LIN {X 0,Y 601.05,Z 422.346,A -85,B 0,C 180,E1 28225.786,E2 28225.786} C_VEL
LIN {X 0,Y 601.044,Z 422.337,A -85,B 0,C 180,E1 28222.492,E2 28222.492} C_VEL
LIN {X 0,Y 601.04,Z 422.335,A -85,B 0,C 180,E1 28219.923,E2 28219.923} C_VEL
LIN {X 0,Y 601.083,Z 422.357,A -85,B 0,C 180,E1 28216.736,E2 28216.736} C_VEL
LIN {X 0,Y 601.144,Z 422.564,A -85,B 0,C 180,E1 28214.936,E2 28214.936} C_VEL
LIN {X 0,Y 604.045,Z 429.719,A -85,B 0,C 180,E1 28213.94,E2 28213.94} C_VEL
LIN {X 0,Y 612.426,Z 450.093,A -85,B 0,C 180,E1 28211.32,E2 28211.32} C_VEL
LIN {X 0,Y 619.561,Z 469.104,A -85,B 0,C 180,E1 28209.079,E2 28209.079} C_VEL
LIN {X 0,Y 619.97,Z 470.564,A -85,B 0,C 180,E1 28208.923,E2 28208.923} C_VEL
LIN {X 0,Y 618.198,Z 495.68,A -85,B 0,C 180,E1 28206.964,E2 28206.964} C_VEL
LIN {X 0,Y 624.328,Z 523.905,A -85,B 0,C 180,E1 28206.115,E2 28206.115} C_VEL
LIN {X 0,Y 624.389,Z 528.229,A -85,B 0,C 180,E1 28206.051,E2 28206.051} C_VEL
LIN {X 0,Y 622.576,Z 534.727,A -85,B 0,C 180,E1 28206.091,E2 28206.091} C_VEL
LIN {X 0,Y 619.497,Z 543.485,A -85,B 0,C 180,E1 28206.191,E2 28206.191} C_VEL
LIN {X 0,Y 618.976,Z 547.292,A -85,B 0,C 180,E1 28206.176,E2 28206.176} C_VEL
LIN {X 0,Y 614.774,Z 810.927,A -85,B 0,C 180,E1 28202.873,E2 28202.873} C_VEL
LIN {X 0,Y 613.983,Z 851.148,A -85,B 0,C 180,E1 28202.339,E2 28202.339} C_VEL
LIN {X 0,Y 613.023,Z 872.802,A -85,B 0,C 180,E1 28201.895,E2 28201.895} C_VEL
LIN {X 0,Y 611.761,Z 895.07,A -85,B 0,C 180,E1 28201.289,E2 28201.289} C_VEL
LIN {X 0,Y 610.189,Z 916.453,A -85,B 0,C 180,E1 28200.53,E2 28200.53} C_VEL
LIN {X 0,Y 608.411,Z 937.861,A -85,B 0,C 180,E1 28199.6,E2 28199.6} C_VEL
LIN {X 0,Y 606.619,Z 956.702,A -85,B 0,C 180,E1 28198.609,E2 28198.609} C_VEL
LIN {X 0,Y 604.551,Z 976.76,A -85,B 0,C 180,E1 28197.374,E2 28197.374} C_VEL
LIN {X 0,Y 602.523,Z 995.2,A -85,B 0,C 180,E1 28196.036,E2 28196.036} C_VEL
LIN {X 0,Y 600.358,Z 1014.63,A -85,B 0,C 180,E1 28194.396,E2 28194.396} C_VEL
LIN {X 0,Y 598.531,Z 1031.433,A -85,B 0,C 180,E1 28192.756,E2 28192.756} C_VEL
LIN {X 0,Y 596.872,Z 1046.866,A -85,B 0,C 180,E1 28191.008,E2 28191.008} C_VEL
LIN {X 0,Y 595.449,Z 1061.5,A -85,B 0,C 180,E1 28189.114,E2 28189.114} C_VEL
LIN {X 0,Y 594.262,Z 1074.683,A -85,B 0,C 180,E1 28187.117,E2 28187.117} C_VEL
LIN {X 0,Y 593.331,Z 1086.983,A -85,B 0,C 180,E1 28184.942,E2 28184.942} C_VEL
LIN {X 0,Y 592.724,Z 1096.907,A -85,B 0,C 180,E1 28182.866,E2 28182.866} C_VEL
LIN {X 0,Y 592.299,Z 1105.822,A -85,B 0,C 180,E1 28180.603,E2 28180.603} C_VEL
LIN {X 0,Y 592.042,Z 1113.446,A -85,B 0,C 180,E1 28178.156,E2 28178.156} C_VEL
LIN {X 0,Y 591.953,Z 1118.281,A -85,B 0,C 180,E1 28176.109,E2 28176.109} C_VEL
LIN {X 0,Y 591.903,Z 1122.06,A -85,B 0,C 180,E1 28173.778,E2 28173.778} C_VEL
LIN {X 0,Y 591.898,Z 1123.925,A -85,B 0,C 180,E1 28171.742,E2 28171.742} C_VEL
LIN {X 0,Y 591.894,Z 1124.401,A -85,B 0,C 180,E1 28169.516,E2 28169.516} C_VEL
LIN {X 0,Y 591.895,Z 1123.448,A -85,B 0,C 180,E1 28167.483,E2 28167.483} C_VEL
LIN {X 0,Y 591.909,Z 1120.693,A -85,B 0,C 180,E1 28165.155,E2 28165.155} C_VEL
LIN {X 0,Y 591.961,Z 1116.818,A -85,B 0,C 180,E1 28163.112,E2 28163.112} C_VEL
LIN {X 0,Y 592.104,Z 1110.894,A -85,B 0,C 180,E1 28160.866,E2 28160.866} C_VEL
LIN {X 0,Y 592.394,Z 1103.29,A -85,B 0,C 180,E1 28158.61,E2 28158.61} C_VEL
LIN {X 0,Y 592.842,Z 1094.611,A -85,B 0,C 180,E1 28156.541,E2 28156.541} C_VEL
LIN {X 0,Y 593.533,Z 1084.376,A -85,B 0,C 180,E1 28154.463,E2 28154.463} C_VEL
LIN {X 0,Y 594.419,Z 1072.701,A -85,B 0,C 180,E1 28152.476,E2 28152.476} C_VEL
LIN {X 0,Y 595.654,Z 1059.219,A -85,B 0,C 180,E1 28150.485,E2 28150.485} C_VEL
LIN {X 0,Y 597.056,Z 1045.112,A -85,B 0,C 180,E1 28148.69,E2 28148.69} C_VEL
LIN {X 0,Y 598.825,Z 1028.383,A -85,B 0,C 180,E1 28146.844,E2 28146.844} C_VEL
LIN {X 0,Y 600.769,Z 1011.25,A -85,B 0,C 180,E1 28145.202,E2 28145.202} C_VEL
LIN {X 0,Y 602.748,Z 993.069,A -85,B 0,C 180,E1 28143.709,E2 28143.709} C_VEL
LIN {X 0,Y 604.798,Z 974.681,A -85,B 0,C 180,E1 28142.394,E2 28142.394} C_VEL
LIN {X 0,Y 606.783,Z 955.027,A -85,B 0,C 180,E1 28141.206,E2 28141.206} C_VEL
LIN {X 0,Y 608.708,Z 934.494,A -85,B 0,C 180,E1 28140.149,E2 28140.149} C_VEL
LIN {X 0,Y 610.427,Z 913.492,A -85,B 0,C 180,E1 28139.265,E2 28139.265} C_VEL
LIN {X 0,Y 612.059,Z 890.14,A -85,B 0,C 180,E1 28138.475,E2 28138.475} C_VEL
LIN {X 0,Y 613.177,Z 869.724,A -85,B 0,C 180,E1 28137.941,E2 28137.941} C_VEL
LIN {X 0,Y 614.133,Z 844.992,A -85,B 0,C 180,E1 28137.477,E2 28137.477} C_VEL
LIN {X 0,Y 617.7,Z 621.355,A -85,B 0,C 180,E1 28134.667,E2 28134.667} C_VEL
LIN {X 0,Y 619.107,Z 530.98,A -85,B 0,C 180,E1 28133.514,E2 28133.514} C_VEL
LIN {X 0,Y 611.434,Z 494.69,A -85,B 0,C 180,E1 28132.397,E2 28132.397} C_VEL
LIN {X 0,Y 613.03,Z 473.555,A -85,B 0,C 180,E1 28130.709,E2 28130.709} C_VEL
LIN {X 0,Y 605.976,Z 454.567,A -85,B 0,C 180,E1 28128.446,E2 28128.446} C_VEL
LIN {X 0,Y 597.834,Z 434.608,A -85,B 0,C 180,E1 28125.85,E2 28125.85} C_VEL
LIN {X 0,Y 593.852,Z 425.716,A -85,B 0,C 180,E1 28124.597,E2 28124.597} C_VEL
LIN {X 0,Y 593.146,Z 423.487,A -85,B 0,C 180,E1 28124.238,E2 28124.238} C_VEL
LIN {X 0,Y 593.126,Z 423.302,A -85,B 0,C 180,E1 28121.364,E2 28121.364} C_VEL
LIN {X 0,Y 593.115,Z 423.346,A -85,B 0,C 180,E1 28118.067,E2 28118.067} C_VEL
LIN {X 0,Y 593.129,Z 423.304,A -85,B 0,C 180,E1 28115.154,E2 28115.154} C_VEL
LIN {X 0,Y 593.105,Z 423.34,A -85,B 0,C 180,E1 28111.962,E2 28111.962} C_VEL
LIN {X 0,Y 593.118,Z 423.349,A -85,B 0,C 180,E1 28109.157,E2 28109.157} C_VEL
LIN {X 0,Y 593.103,Z 423.347,A -85,B 0,C 180,E1 28105.89,E2 28105.89} C_VEL
LIN {X 0,Y 593.124,Z 423.346,A -85,B 0,C 180,E1 28103.008,E2 28103.008} C_VEL
LIN {X 0,Y 593.113,Z 423.346,A -85,B 0,C 180,E1 28099.807,E2 28099.807} C_VEL
LIN {X 0,Y 593.124,Z 423.335,A -85,B 0,C 180,E1 28096.956,E2 28096.956} C_VEL
LIN {X 0,Y 593.122,Z 423.341,A -85,B 0,C 180,E1 28093.751,E2 28093.751} C_VEL
LIN {X 0,Y 593.131,Z 423.343,A -85,B 0,C 180,E1 28090.883,E2 28090.883} C_VEL
LIN {X 0,Y 593.124,Z 423.336,A -85,B 0,C 180,E1 28087.556,E2 28087.556} C_VEL
LIN {X 0,Y 593.143,Z 423.34,A -85,B 0,C 180,E1 28084.738,E2 28084.738} C_VEL
LIN {X 0,Y 593.131,Z 423.344,A -85,B 0,C 180,E1 28081.449,E2 28081.449} C_VEL
LIN {X 0,Y 593.157,Z 423.328,A -85,B 0,C 180,E1 28078.551,E2 28078.551} C_VEL
LIN {X 0,Y 593.137,Z 423.334,A -85,B 0,C 180,E1 28075.359,E2 28075.359} C_VEL
LIN {X 0,Y 593.176,Z 423.345,A -85,B 0,C 180,E1 28072.347,E2 28072.347} C_VEL
LIN {X 0,Y 593.14,Z 423.337,A -85,B 0,C 180,E1 28069.117,E2 28069.117} C_VEL
LIN {X 0,Y 593.198,Z 423.324,A -85,B 0,C 180,E1 28066.052,E2 28066.052} C_VEL
LIN {X 0,Y 593.145,Z 423.341,A -85,B 0,C 180,E1 28062.906,E2 28062.906} C_VEL
LIN {X 0,Y 593.201,Z 423.339,A -85,B 0,C 180,E1 28059.785,E2 28059.785} C_VEL
LIN {X 0,Y 593.153,Z 423.338,A -85,B 0,C 180,E1 28056.663,E2 28056.663} C_VEL
LIN {X 0,Y 593.198,Z 423.333,A -85,B 0,C 180,E1 28053.469,E2 28053.469} C_VEL
LIN {X 0,Y 593.168,Z 423.332,A -85,B 0,C 180,E1 28050.291,E2 28050.291} C_VEL
LIN {X 0,Y 593.171,Z 423.302,A -85,B 0,C 180,E1 28047.011,E2 28047.011} C_VEL
LIN {X 0,Y 593.194,Z 423.336,A -85,B 0,C 180,E1 28043.844,E2 28043.844} C_VEL
LIN {X 0,Y 593.16,Z 423.296,A -85,B 0,C 180,E1 28040.667,E2 28040.667} C_VEL
LIN {X 0,Y 593.194,Z 423.319,A -85,B 0,C 180,E1 28037.587,E2 28037.587} C_VEL
LIN {X 0,Y 593.202,Z 423.558,A -85,B 0,C 180,E1 28036.492,E2 28036.492} C_VEL
LIN {X 0,Y 596.23,Z 430.677,A -85,B 0,C 180,E1 28035.493,E2 28035.493} C_VEL
LIN {X 0,Y 604.145,Z 449.031,A -85,B 0,C 180,E1 28033.121,E2 28033.121} C_VEL
LIN {X 0,Y 607.608,Z 457.418,A -85,B 0,C 180,E1 28032.136,E2 28032.136} C_VEL
LIN {X 0,Y 620.44,Z 478.904,A -85,B 0,C 180,E1 28030.804,E2 28030.804} C_VEL
LIN {X 0,Y 622.327,Z 489.051,A -85,B 0,C 180,E1 28030.513,E2 28030.513} C_VEL
LIN {X 0,Y 617.253,Z 739.769,A -85,B 0,C 180,E1 28027.182,E2 28027.182} C_VEL
LIN {X 0,Y 615.172,Z 843.964,A -85,B 0,C 180,E1 28025.791,E2 28025.791} C_VEL
LIN {X 0,Y 614.103,Z 869.036,A -85,B 0,C 180,E1 28025.297,E2 28025.297} C_VEL
LIN {X 0,Y 612.948,Z 889.774,A -85,B 0,C 180,E1 28024.756,E2 28024.756} C_VEL
LIN {X 0,Y 611.336,Z 914.776,A -85,B 0,C 180,E1 28023.93,E2 28023.93} C_VEL
LIN {X 0,Y 609.706,Z 936.084,A -85,B 0,C 180,E1 28023.068,E2 28023.068} C_VEL
LIN {X 0,Y 607.878,Z 958.694,A -85,B 0,C 180,E1 28021.982,E2 28021.982} C_VEL
LIN {X 0,Y 606.11,Z 978.363,A -85,B 0,C 180,E1 28020.868,E2 28020.868} C_VEL
LIN {X 0,Y 604.212,Z 998.769,A -85,B 0,C 180,E1 28019.548,E2 28019.548} C_VEL
LIN {X 0,Y 602.242,Z 1018.444,A -85,B 0,C 180,E1 28018.065,E2 28018.065} C_VEL
LIN {X 0,Y 600.563,Z 1035.551,A -85,B 0,C 180,E1 28016.607,E2 28016.607} C_VEL
LIN {X 0,Y 598.715,Z 1054.222,A -85,B 0,C 180,E1 28014.783,E2 28014.783} C_VEL
LIN {X 0,Y 597.317,Z 1068.791,A -85,B 0,C 180,E1 28013.165,E2 28013.165} C_VEL
LIN {X 0,Y 595.868,Z 1084.777,A -85,B 0,C 180,E1 28011.148,E2 28011.148} C_VEL
LIN {X 0,Y 594.797,Z 1097.221,A -85,B 0,C 180,E1 28009.34,E2 28009.34} C_VEL
LIN {X 0,Y 593.82,Z 1109.687,A -85,B 0,C 180,E1 28007.239,E2 28007.239} C_VEL
LIN {X 0,Y 593.064,Z 1120.636,A -85,B 0,C 180,E1 28005.049,E2 28005.049} C_VEL
LIN {X 0,Y 592.573,Z 1129.582,A -85,B 0,C 180,E1 28002.969,E2 28002.969} C_VEL
LIN {X 0,Y 592.216,Z 1137.906,A -85,B 0,C 180,E1 28000.605,E2 28000.605} C_VEL
LIN {X 0,Y 592.035,Z 1143.491,A -85,B 0,C 180,E1 27998.645,E2 27998.645} C_VEL
LIN {X 0,Y 591.95,Z 1148.695,A -85,B 0,C 180,E1 27996.304,E2 27996.304} C_VEL
LIN {X 0,Y 591.92,Z 1152.008,A -85,B 0,C 180,E1 27994.068,E2 27994.068} C_VEL
LIN {X 0,Y 591.908,Z 1153.903,A -85,B 0,C 180,E1 27991.936,E2 27991.936} C_VEL
LIN {X 0,Y 591.885,Z 1154.394,A -85,B 0,C 180,E1 27989.516,E2 27989.516} C_VEL
LIN {X 0,Y 591.897,Z 1153.494,A -85,B 0,C 180,E1 27987.483,E2 27987.483} C_VEL
LIN {X 0,Y 591.911,Z 1151.085,A -85,B 0,C 180,E1 27985.155,E2 27985.155} C_VEL
LIN {X 0,Y 591.973,Z 1147.102,A -85,B 0,C 180,E1 27982.917,E2 27982.917} C_VEL
LIN {X 0,Y 592.066,Z 1142.219,A -85,B 0,C 180,E1 27980.866,E2 27980.866} C_VEL
LIN {X 0,Y 592.321,Z 1134.659,A -85,B 0,C 180,E1 27978.411,E2 27978.411} C_VEL
LIN {X 0,Y 592.678,Z 1127.151,A -85,B 0,C 180,E1 27976.438,E2 27976.438} C_VEL
LIN {X 0,Y 593.285,Z 1117.27,A -85,B 0,C 180,E1 27974.225,E2 27974.225} C_VEL
LIN {X 0,Y 594.113,Z 1105.682,A -85,B 0,C 180,E1 27972.062,E2 27972.062} C_VEL
LIN {X 0,Y 595.031,Z 1094.406,A -85,B 0,C 180,E1 27970.225,E2 27970.225} C_VEL
LIN {X 0,Y 596.331,Z 1079.433,A -85,B 0,C 180,E1 27968.146,E2 27968.146} C_VEL
LIN {X 0,Y 597.651,Z 1065.334,A -85,B 0,C 180,E1 27966.431,E2 27966.431} C_VEL
LIN {X 0,Y 599.431,Z 1047.001,A -85,B 0,C 180,E1 27964.479,E2 27964.479} C_VEL
LIN {X 0,Y 601.065,Z 1030.416,A -85,B 0,C 180,E1 27962.936,E2 27962.936} C_VEL
LIN {X 0,Y 603.114,Z 1009.862,A -85,B 0,C 180,E1 27961.263,E2 27961.263} C_VEL
LIN {X 0,Y 604.896,Z 991.183,A -85,B 0,C 180,E1 27959.943,E2 27959.943} C_VEL
LIN {X 0,Y 606.901,Z 969.837,A -85,B 0,C 180,E1 27958.626,E2 27958.626} C_VEL
LIN {X 0,Y 608.666,Z 949.321,A -85,B 0,C 180,E1 27957.549,E2 27957.549} C_VEL
LIN {X 0,Y 610.346,Z 928.452,A -85,B 0,C 180,E1 27956.602,E2 27956.602} C_VEL
LIN {X 0,Y 611.969,Z 905.031,A -85,B 0,C 180,E1 27955.725,E2 27955.725} C_VEL
LIN {X 0,Y 613.339,Z 882.784,A -85,B 0,C 180,E1 27955.043,E2 27955.043} C_VEL
LIN {X 0,Y 614.638,Z 857.534,A -85,B 0,C 180,E1 27954.456,E2 27954.456} C_VEL
LIN {X 0,Y 615.43,Z 835.19,A -85,B 0,C 180,E1 27954.079,E2 27954.079} C_VEL
LIN {X 0,Y 620.145,Z 592.09,A -85,B 0,C 180,E1 27950.858,E2 27950.858} C_VEL
LIN {X 0,Y 622.173,Z 487.31,A -85,B 0,C 180,E1 27949.452,E2 27949.452} C_VEL
LIN {X 0,Y 620.052,Z 478.166,A -85,B 0,C 180,E1 27949.158,E2 27949.158} C_VEL
LIN {X 0,Y 607.39,Z 457,A -85,B 0,C 180,E1 27947.835,E2 27947.835} C_VEL
LIN {X 0,Y 599.631,Z 438.401,A -85,B 0,C 180,E1 27945.537,E2 27945.537} C_VEL
LIN {X 0,Y 594.136,Z 426.221,A -85,B 0,C 180,E1 27943.898,E2 27943.898} C_VEL
LIN {X 0,Y 593.189,Z 423.473,A -85,B 0,C 180,E1 27943.481,E2 27943.481} C_VEL
LIN {X 0,Y 593.196,Z 423.3,A -85,B 0,C 180,E1 27940.21,E2 27940.21} C_VEL
LIN {X 0,Y 593.185,Z 423.342,A -85,B 0,C 180,E1 27936.966,E2 27936.966} C_VEL
LIN {X 0,Y 593.163,Z 423.294,A -85,B 0,C 180,E1 27933.683,E2 27933.683} C_VEL
LIN {X 0,Y 593.2,Z 423.341,A -85,B 0,C 180,E1 27930.488,E2 27930.488} C_VEL
LIN {X 0,Y 593.157,Z 423.342,A -85,B 0,C 180,E1 27927.291,E2 27927.291} C_VEL
LIN {X 0,Y 593.2,Z 423.34,A -85,B 0,C 180,E1 27924.074,E2 27924.074} C_VEL
LIN {X 0,Y 593.156,Z 423.339,A -85,B 0,C 180,E1 27920.939,E2 27920.939} C_VEL
LIN {X 0,Y 593.172,Z 423.331,A -85,B 0,C 180,E1 27917.663,E2 27917.663} C_VEL
LIN {X 0,Y 593.162,Z 423.331,A -85,B 0,C 180,E1 27914.626,E2 27914.626} C_VEL
LIN {X 0,Y 593.153,Z 423.339,A -85,B 0,C 180,E1 27911.375,E2 27911.375} C_VEL
LIN {X 0,Y 593.177,Z 423.336,A -85,B 0,C 180,E1 27908.317,E2 27908.317} C_VEL
LIN {X 0,Y 593.138,Z 423.332,A -85,B 0,C 180,E1 27905.126,E2 27905.126} C_VEL
LIN {X 0,Y 593.189,Z 423.336,A -85,B 0,C 180,E1 27902.029,E2 27902.029} C_VEL
LIN {X 0,Y 593.132,Z 423.345,A -85,B 0,C 180,E1 27898.937,E2 27898.937} C_VEL
LIN {X 0,Y 593.19,Z 423.323,A -85,B 0,C 180,E1 27895.843,E2 27895.843} C_VEL
LIN {X 0,Y 593.121,Z 423.337,A -85,B 0,C 180,E1 27892.736,E2 27892.736} C_VEL
LIN {X 0,Y 593.192,Z 423.343,A -85,B 0,C 180,E1 27889.609,E2 27889.609} C_VEL
LIN {X 0,Y 593.115,Z 423.34,A -85,B 0,C 180,E1 27886.547,E2 27886.547} C_VEL
LIN {X 0,Y 593.188,Z 423.328,A -85,B 0,C 180,E1 27883.55,E2 27883.55} C_VEL
LIN {X 0,Y 593.11,Z 423.345,A -85,B 0,C 180,E1 27880.457,E2 27880.457} C_VEL
LIN {X 0,Y 593.188,Z 423.342,A -85,B 0,C 180,E1 27877.398,E2 27877.398} C_VEL
LIN {X 0,Y 593.103,Z 423.345,A -85,B 0,C 180,E1 27874.325,E2 27874.325} C_VEL
LIN {X 0,Y 593.163,Z 423.335,A -85,B 0,C 180,E1 27871.177,E2 27871.177} C_VEL
LIN {X 0,Y 593.093,Z 423.339,A -85,B 0,C 180,E1 27868.264,E2 27868.264} C_VEL
LIN {X 0,Y 593.159,Z 423.309,A -85,B 0,C 180,E1 27865.148,E2 27865.148} C_VEL
LIN {X 0,Y 593.097,Z 423.339,A -85,B 0,C 180,E1 27862.092,E2 27862.092} C_VEL
LIN {X 0,Y 593.171,Z 423.297,A -85,B 0,C 180,E1 27859.025,E2 27859.025} C_VEL
LIN {X 0,Y 593.105,Z 423.337,A -85,B 0,C 180,E1 27856.006,E2 27856.006} C_VEL
LIN {X 0,Y 593.191,Z 423.746,A -85,B 0,C 180,E1 27855.582,E2 27855.582} C_VEL
LIN {X 0,Y 601.081,Z 442.504,A -85,B 0,C 180,E1 27853.003,E2 27853.003} C_VEL
LIN {X 0,Y 607.647,Z 459.038,A -85,B 0,C 180,E1 27850.913,E2 27850.913} C_VEL
LIN {X 0,Y 613.042,Z 474.205,A -85,B 0,C 180,E1 27849.14,E2 27849.14} C_VEL
LIN {X 0,Y 611.468,Z 495.318,A -85,B 0,C 180,E1 27847.48,E2 27847.48} C_VEL
LIN {X 0,Y 619.238,Z 532.257,A -85,B 0,C 180,E1 27846.367,E2 27846.367} C_VEL
LIN {X 0,Y 618.976,Z 547.292,A -85,B 0,C 180,E1 27846.176,E2 27846.176} C_VEL
LIN {X 0,Y 618.033,Z 554.991,A -85,B 0,C 180,E1 27846.136,E2 27846.136} C_VEL
LIN {X 0,Y 612.713,Z 575.535,A -85,B 0,C 180,E1 27846.236,E2 27846.236} C_VEL
LIN {X 0,Y 612.009,Z 582.141,A -85,B 0,C 180,E1 27846.195,E2 27846.195} C_VEL
LIN {X 0,Y 607.943,Z 828.787,A -85,B 0,C 180,E1 27843.084,E2 27843.084} C_VEL
LIN {X 0,Y 607.185,Z 856.005,A -85,B 0,C 180,E1 27842.679,E2 27842.679} C_VEL
LIN {X 0,Y 606.22,Z 876.458,A -85,B 0,C 180,E1 27842.237,E2 27842.237} C_VEL
LIN {X 0,Y 604.704,Z 899.838,A -85,B 0,C 180,E1 27841.557,E2 27841.557} C_VEL
LIN {X 0,Y 603.091,Z 921.266,A -85,B 0,C 180,E1 27840.762,E2 27840.762} C_VEL
LIN {X 0,Y 601.196,Z 941.808,A -85,B 0,C 180,E1 27839.821,E2 27839.821} C_VEL
LIN {X 0,Y 599.287,Z 961.134,A -85,B 0,C 180,E1 27838.774,E2 27838.774} C_VEL
LIN {X 0,Y 597.129,Z 980.515,A -85,B 0,C 180,E1 27837.527,E2 27837.527} C_VEL
LIN {X 0,Y 595.111,Z 998.251,A -85,B 0,C 180,E1 27836.205,E2 27836.205} C_VEL
LIN {X 0,Y 592.941,Z 1016.199,A -85,B 0,C 180,E1 27834.642,E2 27834.642} C_VEL
LIN {X 0,Y 591.03,Z 1032.627,A -85,B 0,C 180,E1 27833.004,E2 27833.004} C_VEL
LIN {X 0,Y 589.218,Z 1048.24,A -85,B 0,C 180,E1 27831.19,E2 27831.19} C_VEL
LIN {X 0,Y 587.627,Z 1063.346,A -85,B 0,C 180,E1 27829.172,E2 27829.172} C_VEL
LIN {X 0,Y 586.448,Z 1075.686,A -85,B 0,C 180,E1 27827.258,E2 27827.258} C_VEL
LIN {X 0,Y 585.481,Z 1087.333,A -85,B 0,C 180,E1 27825.147,E2 27825.147} C_VEL
LIN {X 0,Y 584.821,Z 1097.227,A -85,B 0,C 180,E1 27823.043,E2 27823.043} C_VEL
LIN {X 0,Y 584.358,Z 1105.737,A -85,B 0,C 180,E1 27820.835,E2 27820.835} C_VEL
LIN {X 0,Y 584.091,Z 1112.836,A -85,B 0,C 180,E1 27818.565,E2 27818.565} C_VEL
LIN {X 0,Y 583.959,Z 1117.726,A -85,B 0,C 180,E1 27816.489,E2 27816.489} C_VEL
LIN {X 0,Y 583.915,Z 1121.617,A -85,B 0,C 180,E1 27814.223,E2 27814.223} C_VEL
LIN {X 0,Y 583.907,Z 1123.814,A -85,B 0,C 180,E1 27811.963,E2 27811.963} C_VEL
LIN {X 0,Y 583.896,Z 1124.423,A -85,B 0,C 180,E1 27809.608,E2 27809.608} C_VEL
LIN {X 0,Y 583.896,Z 1123.546,A -85,B 0,C 180,E1 27807.546,E2 27807.546} C_VEL
LIN {X 0,Y 583.907,Z 1121.046,A -85,B 0,C 180,E1 27805.285,E2 27805.285} C_VEL
LIN {X 0,Y 583.961,Z 1117.301,A -85,B 0,C 180,E1 27803.215,E2 27803.215} C_VEL
LIN {X 0,Y 584.112,Z 1111.675,A -85,B 0,C 180,E1 27800.939,E2 27800.939} C_VEL
LIN {X 0,Y 584.384,Z 1104.957,A -85,B 0,C 180,E1 27798.852,E2 27798.852} C_VEL
LIN {X 0,Y 584.895,Z 1095.828,A -85,B 0,C 180,E1 27796.556,E2 27796.556} C_VEL
LIN {X 0,Y 585.614,Z 1085.762,A -85,B 0,C 180,E1 27794.451,E2 27794.451} C_VEL
LIN {X 0,Y 586.614,Z 1073.704,A -85,B 0,C 180,E1 27792.331,E2 27792.331} C_VEL
LIN {X 0,Y 587.932,Z 1060.467,A -85,B 0,C 180,E1 27790.322,E2 27790.322} C_VEL
LIN {X 0,Y 589.413,Z 1046.487,A -85,B 0,C 180,E1 27788.504,E2 27788.504} C_VEL
LIN {X 0,Y 591.259,Z 1030.422,A -85,B 0,C 180,E1 27786.676,E2 27786.676} C_VEL
LIN {X 0,Y 593.201,Z 1014.112,A -85,B 0,C 180,E1 27785.074,E2 27785.074} C_VEL
LIN {X 0,Y 595.475,Z 994.847,A -85,B 0,C 180,E1 27783.439,E2 27783.439} C_VEL
LIN {X 0,Y 597.502,Z 977.421,A -85,B 0,C 180,E1 27782.167,E2 27782.167} C_VEL
LIN {X 0,Y 599.666,Z 957.308,A -85,B 0,C 180,E1 27780.918,E2 27780.918} C_VEL
LIN {X 0,Y 601.526,Z 938.496,A -85,B 0,C 180,E1 27779.922,E2 27779.922} C_VEL
LIN {X 0,Y 603.405,Z 917.009,A -85,B 0,C 180,E1 27778.979,E2 27778.979} C_VEL
LIN {X 0,Y 604.985,Z 896.363,A -85,B 0,C 180,E1 27778.237,E2 27778.237} C_VEL
LIN {X 0,Y 606.369,Z 873.599,A -85,B 0,C 180,E1 27777.604,E2 27777.604} C_VEL
LIN {X 0,Y 607.34,Z 852.734,A -85,B 0,C 180,E1 27777.169,E2 27777.169} C_VEL
LIN {X 0,Y 608.099,Z 819.646,A -85,B 0,C 180,E1 27776.711,E2 27776.711} C_VEL
LIN {X 0,Y 612.468,Z 559.419,A -85,B 0,C 180,E1 27773.426,E2 27773.426} C_VEL
LIN {X 0,Y 612.791,Z 532.472,A -85,B 0,C 180,E1 27773.066,E2 27773.066} C_VEL
LIN {X 0,Y 604.761,Z 494.235,A -85,B 0,C 180,E1 27771.864,E2 27771.864} C_VEL
LIN {X 0,Y 606.055,Z 476.769,A -85,B 0,C 180,E1 27770.443,E2 27770.443} C_VEL
LIN {X 0,Y 599.286,Z 458.457,A -85,B 0,C 180,E1 27768.229,E2 27768.229} C_VEL
LIN {X 0,Y 591.613,Z 439.49,A -85,B 0,C 180,E1 27765.732,E2 27765.732} C_VEL
LIN {X 0,Y 586.509,Z 427.857,A -85,B 0,C 180,E1 27764.073,E2 27764.073} C_VEL
LIN {X 0,Y 585.209,Z 424.511,A -85,B 0,C 180,E1 27763.554,E2 27763.554} C_VEL
LIN {X 0,Y 585.206,Z 424.291,A -85,B 0,C 180,E1 27760.487,E2 27760.487} C_VEL
LIN {X 0,Y 585.166,Z 424.319,A -85,B 0,C 180,E1 27757.707,E2 27757.707} C_VEL
LIN {X 0,Y 585.222,Z 424.301,A -85,B 0,C 180,E1 27754.558,E2 27754.558} C_VEL
LIN {X 0,Y 585.162,Z 424.327,A -85,B 0,C 180,E1 27751.525,E2 27751.525} C_VEL
LIN {X 0,Y 585.203,Z 424.323,A -85,B 0,C 180,E1 27748.359,E2 27748.359} C_VEL
LIN {X 0,Y 585.159,Z 424.335,A -85,B 0,C 180,E1 27745.398,E2 27745.398} C_VEL
LIN {X 0,Y 585.197,Z 424.331,A -85,B 0,C 180,E1 27742.167,E2 27742.167} C_VEL
LIN {X 0,Y 585.17,Z 424.335,A -85,B 0,C 180,E1 27739.256,E2 27739.256} C_VEL
LIN {X 0,Y 585.196,Z 424.328,A -85,B 0,C 180,E1 27735.968,E2 27735.968} C_VEL
LIN {X 0,Y 585.178,Z 424.327,A -85,B 0,C 180,E1 27733.104,E2 27733.104} C_VEL
LIN {X 0,Y 585.201,Z 424.33,A -85,B 0,C 180,E1 27729.838,E2 27729.838} C_VEL
LIN {X 0,Y 585.19,Z 424.326,A -85,B 0,C 180,E1 27726.91,E2 27726.91} C_VEL
LIN {X 0,Y 585.191,Z 424.317,A -85,B 0,C 180,E1 27723.527,E2 27723.527} C_VEL
LIN {X 0,Y 585.217,Z 424.331,A -85,B 0,C 180,E1 27720.587,E2 27720.587} C_VEL
LIN {X 0,Y 585.196,Z 424.332,A -85,B 0,C 180,E1 27717.356,E2 27717.356} C_VEL
LIN {X 0,Y 585.25,Z 424.314,A -85,B 0,C 180,E1 27714.215,E2 27714.215} C_VEL
LIN {X 0,Y 585.199,Z 424.328,A -85,B 0,C 180,E1 27711.154,E2 27711.154} C_VEL
LIN {X 0,Y 585.262,Z 424.329,A -85,B 0,C 180,E1 27707.97,E2 27707.97} C_VEL
LIN {X 0,Y 585.203,Z 424.324,A -85,B 0,C 180,E1 27704.846,E2 27704.846} C_VEL
LIN {X 0,Y 585.256,Z 424.312,A -85,B 0,C 180,E1 27701.678,E2 27701.678} C_VEL
LIN {X 0,Y 585.217,Z 424.325,A -85,B 0,C 180,E1 27698.553,E2 27698.553} C_VEL
LIN {X 0,Y 585.238,Z 424.324,A -85,B 0,C 180,E1 27695.254,E2 27695.254} C_VEL
LIN {X 0,Y 585.255,Z 424.328,A -85,B 0,C 180,E1 27692.041,E2 27692.041} C_VEL
LIN {X 0,Y 585.225,Z 424.332,A -85,B 0,C 180,E1 27688.822,E2 27688.822} C_VEL
LIN {X 0,Y 585.253,Z 424.279,A -85,B 0,C 180,E1 27685.609,E2 27685.609} C_VEL
LIN {X 0,Y 585.225,Z 424.316,A -85,B 0,C 180,E1 27682.414,E2 27682.414} C_VEL
LIN {X 0,Y 585.258,Z 424.302,A -85,B 0,C 180,E1 27679.187,E2 27679.187} C_VEL
LIN {X 0,Y 585.292,Z 424.566,A -85,B 0,C 180,E1 27677.198,E2 27677.198} C_VEL
LIN {X 0,Y 588.532,Z 432.056,A -85,B 0,C 180,E1 27676.118,E2 27676.118} C_VEL
LIN {X 0,Y 596.656,Z 450.909,A -85,B 0,C 180,E1 27673.618,E2 27673.618} C_VEL
LIN {X 0,Y 599.594,Z 457.875,A -85,B 0,C 180,E1 27672.78,E2 27672.78} C_VEL
LIN {X 0,Y 614.47,Z 482.491,A -85,B 0,C 180,E1 27671.201,E2 27671.201} C_VEL
LIN {X 0,Y 616.048,Z 490.662,A -85,B 0,C 180,E1 27670.957,E2 27670.957} C_VEL
LIN {X 0,Y 610.694,Z 740.474,A -85,B 0,C 180,E1 27667.605,E2 27667.605} C_VEL
LIN {X 0,Y 608.499,Z 843.797,A -85,B 0,C 180,E1 27666.209,E2 27666.209} C_VEL
LIN {X 0,Y 607.364,Z 868.981,A -85,B 0,C 180,E1 27665.708,E2 27665.708} C_VEL
LIN {X 0,Y 606.136,Z 889.862,A -85,B 0,C 180,E1 27665.157,E2 27665.157} C_VEL
LIN {X 0,Y 604.457,Z 914.363,A -85,B 0,C 180,E1 27664.339,E2 27664.339} C_VEL
LIN {X 0,Y 602.732,Z 935.519,A -85,B 0,C 180,E1 27663.471,E2 27663.471} C_VEL
LIN {X 0,Y 600.762,Z 958.317,A -85,B 0,C 180,E1 27662.365,E2 27662.365} C_VEL
LIN {X 0,Y 598.876,Z 978.222,A -85,B 0,C 180,E1 27661.226,E2 27661.226} C_VEL
LIN {X 0,Y 596.875,Z 998.757,A -85,B 0,C 180,E1 27659.883,E2 27659.883} C_VEL
LIN {X 0,Y 594.831,Z 1018.144,A -85,B 0,C 180,E1 27658.406,E2 27658.406} C_VEL
LIN {X 0,Y 593.03,Z 1035.419,A -85,B 0,C 180,E1 27656.918,E2 27656.918} C_VEL
LIN {X 0,Y 591.107,Z 1053.935,A -85,B 0,C 180,E1 27655.088,E2 27655.088} C_VEL
LIN {X 0,Y 589.619,Z 1068.567,A -85,B 0,C 180,E1 27653.444,E2 27653.444} C_VEL
LIN {X 0,Y 588.12,Z 1084.292,A -85,B 0,C 180,E1 27651.44,E2 27651.44} C_VEL
LIN {X 0,Y 586.969,Z 1096.798,A -85,B 0,C 180,E1 27649.605,E2 27649.605} C_VEL
LIN {X 0,Y 586.005,Z 1108.975,A -85,B 0,C 180,E1 27647.579,E2 27647.579} C_VEL
LIN {X 0,Y 585.225,Z 1119.717,A -85,B 0,C 180,E1 27645.458,E2 27645.458} C_VEL
LIN {X 0,Y 584.68,Z 1128.366,A -85,B 0,C 180,E1 27643.449,E2 27643.449} C_VEL
LIN {X 0,Y 584.267,Z 1136.997,A -85,B 0,C 180,E1 27641.05,E2 27641.05} C_VEL
LIN {X 0,Y 584.053,Z 1143.012,A -85,B 0,C 180,E1 27638.951,E2 27638.951} C_VEL
LIN {X 0,Y 583.962,Z 1147.928,A -85,B 0,C 180,E1 27636.785,E2 27636.785} C_VEL
LIN {X 0,Y 583.924,Z 1151.781,A -85,B 0,C 180,E1 27634.321,E2 27634.321} C_VEL
LIN {X 0,Y 583.91,Z 1153.698,A -85,B 0,C 180,E1 27632.257,E2 27632.257} C_VEL
LIN {X 0,Y 583.903,Z 1154.484,A -85,B 0,C 180,E1 27629.902,E2 27629.902} C_VEL
LIN {X 0,Y 583.906,Z 1153.63,A -85,B 0,C 180,E1 27627.645,E2 27627.645} C_VEL
LIN {X 0,Y 583.924,Z 1151.666,A -85,B 0,C 180,E1 27625.581,E2 27625.581} C_VEL
LIN {X 0,Y 583.969,Z 1147.721,A -85,B 0,C 180,E1 27623.116,E2 27623.116} C_VEL
LIN {X 0,Y 584.054,Z 1142.982,A -85,B 0,C 180,E1 27621.037,E2 27621.037} C_VEL
LIN {X 0,Y 584.278,Z 1136.692,A -85,B 0,C 180,E1 27618.85,E2 27618.85} C_VEL
LIN {X 0,Y 584.68,Z 1128.365,A -85,B 0,C 180,E1 27616.551,E2 27616.551} C_VEL
LIN {X 0,Y 585.225,Z 1119.721,A -85,B 0,C 180,E1 27614.542,E2 27614.542} C_VEL
LIN {X 0,Y 586.006,Z 1108.984,A -85,B 0,C 180,E1 27612.421,E2 27612.421} C_VEL
LIN {X 0,Y 586.972,Z 1096.79,A -85,B 0,C 180,E1 27610.392,E2 27610.392} C_VEL
LIN {X 0,Y 588.263,Z 1082.853,A -85,B 0,C 180,E1 27608.356,E2 27608.356} C_VEL
LIN {X 0,Y 589.741,Z 1067.383,A -85,B 0,C 180,E1 27606.413,E2 27606.413} C_VEL
LIN {X 0,Y 591.461,Z 1050.759,A -85,B 0,C 180,E1 27604.57,E2 27604.57} C_VEL
LIN {X 0,Y 593.32,Z 1032.57,A -85,B 0,C 180,E1 27602.825,E2 27602.825} C_VEL
LIN {X 0,Y 595.296,Z 1014.006,A -85,B 0,C 180,E1 27601.257,E2 27601.257} C_VEL
LIN {X 0,Y 597.38,Z 993.315,A -85,B 0,C 180,E1 27599.747,E2 27599.747} C_VEL
LIN {X 0,Y 599.331,Z 973.55,A -85,B 0,C 180,E1 27598.488,E2 27598.488} C_VEL
LIN {X 0,Y 601.394,Z 951.267,A -85,B 0,C 180,E1 27597.277,E2 27597.277} C_VEL
LIN {X 0,Y 603.047,Z 931.944,A -85,B 0,C 180,E1 27596.372,E2 27596.372} C_VEL
LIN {X 0,Y 604.917,Z 907.935,A -85,B 0,C 180,E1 27595.427,E2 27595.427} C_VEL
LIN {X 0,Y 606.352,Z 886.082,A -85,B 0,C 180,E1 27594.733,E2 27594.733} C_VEL
LIN {X 0,Y 607.734,Z 861.727,A -85,B 0,C 180,E1 27594.124,E2 27594.124} C_VEL
LIN {X 0,Y 608.676,Z 838.024,A -85,B 0,C 180,E1 27593.704,E2 27593.704} C_VEL
LIN {X 0,Y 613.716,Z 595.078,A -85,B 0,C 180,E1 27590.446,E2 27590.446} C_VEL
LIN {X 0,Y 615.899,Z 489.034,A -85,B 0,C 180,E1 27589.009,E2 27589.009} C_VEL
LIN {X 0,Y 614.289,Z 482.177,A -85,B 0,C 180,E1 27588.783,E2 27588.783} C_VEL
LIN {X 0,Y 599.373,Z 457.442,A -85,B 0,C 180,E1 27587.19,E2 27587.19} C_VEL
LIN {X 0,Y 591.875,Z 439.643,A -85,B 0,C 180,E1 27584.923,E2 27584.923} C_VEL
LIN {X 0,Y 586.099,Z 427.026,A -85,B 0,C 180,E1 27583.166,E2 27583.166} C_VEL
LIN {X 0,Y 585.276,Z 424.463,A -85,B 0,C 180,E1 27582.766,E2 27582.766} C_VEL
LIN {X 0,Y 585.222,Z 424.283,A -85,B 0,C 180,E1 27579.591,E2 27579.591} C_VEL
LIN {X 0,Y 585.258,Z 424.329,A -85,B 0,C 180,E1 27576.359,E2 27576.359} C_VEL
LIN {X 0,Y 585.224,Z 424.287,A -85,B 0,C 180,E1 27573.144,E2 27573.144} C_VEL
LIN {X 0,Y 585.24,Z 424.32,A -85,B 0,C 180,E1 27569.814,E2 27569.814} C_VEL
LIN {X 0,Y 585.254,Z 424.323,A -85,B 0,C 180,E1 27566.591,E2 27566.591} C_VEL
LIN {X 0,Y 585.215,Z 424.327,A -85,B 0,C 180,E1 27563.353,E2 27563.353} C_VEL
LIN {X 0,Y 585.262,Z 424.328,A -85,B 0,C 180,E1 27560.188,E2 27560.188} C_VEL
LIN {X 0,Y 585.211,Z 424.329,A -85,B 0,C 180,E1 27556.988,E2 27556.988} C_VEL
LIN {X 0,Y 585.243,Z 424.316,A -85,B 0,C 180,E1 27553.738,E2 27553.738} C_VEL
LIN {X 0,Y 585.215,Z 424.324,A -85,B 0,C 180,E1 27550.634,E2 27550.634} C_VEL
LIN {X 0,Y 585.208,Z 424.331,A -85,B 0,C 180,E1 27547.264,E2 27547.264} C_VEL
LIN {X 0,Y 585.237,Z 424.321,A -85,B 0,C 180,E1 27544.213,E2 27544.213} C_VEL
LIN {X 0,Y 585.192,Z 424.316,A -85,B 0,C 180,E1 27540.979,E2 27540.979} C_VEL
LIN {X 0,Y 585.251,Z 424.33,A -85,B 0,C 180,E1 27537.944,E2 27537.944} C_VEL
LIN {X 0,Y 585.186,Z 424.333,A -85,B 0,C 180,E1 27534.804,E2 27534.804} C_VEL
LIN {X 0,Y 585.256,Z 424.311,A -85,B 0,C 180,E1 27531.749,E2 27531.749} C_VEL
LIN {X 0,Y 585.18,Z 424.33,A -85,B 0,C 180,E1 27528.668,E2 27528.668} C_VEL
LIN {X 0,Y 585.262,Z 424.328,A -85,B 0,C 180,E1 27525.556,E2 27525.556} C_VEL
LIN {X 0,Y 585.174,Z 424.328,A -85,B 0,C 180,E1 27522.396,E2 27522.396} C_VEL
LIN {X 0,Y 585.228,Z 424.318,A -85,B 0,C 180,E1 27519.288,E2 27519.288} C_VEL
LIN {X 0,Y 585.167,Z 424.334,A -85,B 0,C 180,E1 27516.325,E2 27516.325} C_VEL
LIN {X 0,Y 585.223,Z 424.331,A -85,B 0,C 180,E1 27513.188,E2 27513.188} C_VEL
LIN {X 0,Y 585.161,Z 424.339,A -85,B 0,C 180,E1 27510.182,E2 27510.182} C_VEL
LIN {X 0,Y 585.208,Z 424.338,A -85,B 0,C 180,E1 27507.027,E2 27507.027} C_VEL
LIN {X 0,Y 585.155,Z 424.287,A -85,B 0,C 180,E1 27503.998,E2 27503.998} C_VEL
LIN {X 0,Y 585.189,Z 424.332,A -85,B 0,C 180,E1 27500.717,E2 27500.717} C_VEL
LIN {X 0,Y 585.168,Z 424.3,A -85,B 0,C 180,E1 27497.815,E2 27497.815} C_VEL
LIN {X 0,Y 585.215,Z 424.639,A -85,B 0,C 180,E1 27496.311,E2 27496.311} C_VEL
LIN {X 0,Y 591.796,Z 439.991,A -85,B 0,C 180,E1 27494.104,E2 27494.104} C_VEL
LIN {X 0,Y 599.538,Z 459.161,A -85,B 0,C 180,E1 27491.588,E2 27491.588} C_VEL
LIN {X 0,Y 606.167,Z 477.085,A -85,B 0,C 180,E1 27489.425,E2 27489.425} C_VEL
LIN {X 0,Y 604.789,Z 494.954,A -85,B 0,C 180,E1 27488.007,E2 27488.007} C_VEL
LIN {X 0,Y 612.934,Z 533.817,A -85,B 0,C 180,E1 27486.811,E2 27486.811} C_VEL
LIN {X 0,Y 612.009,Z 582.141,A -85,B 0,C 180,E1 27486.195,E2 27486.195} C_VEL
LIN {X 0,Y 611.086,Z 589.841,A -85,B 0,C 180,E1 27486.154,E2 27486.154} C_VEL
LIN {X 0,Y 605.761,Z 610.388,A -85,B 0,C 180,E1 27486.258,E2 27486.258} C_VEL
LIN {X 0,Y 605.065,Z 616.995,A -85,B 0,C 180,E1 27486.217,E2 27486.217} C_VEL
LIN {X 0,Y 601.034,Z 844.483,A -85,B 0,C 180,E1 27483.311,E2 27483.311} C_VEL
LIN {X 0,Y 600.031,Z 868.599,A -85,B 0,C 180,E1 27482.861,E2 27482.861} C_VEL
LIN {X 0,Y 598.803,Z 889.331,A -85,B 0,C 180,E1 27482.319,E2 27482.319} C_VEL
LIN {X 0,Y 597.133,Z 911.847,A -85,B 0,C 180,E1 27481.56,E2 27481.56} C_VEL
LIN {X 0,Y 595.384,Z 931.37,A -85,B 0,C 180,E1 27480.744,E2 27480.744} C_VEL
LIN {X 0,Y 593.105,Z 953.929,A -85,B 0,C 180,E1 27479.601,E2 27479.601} C_VEL
LIN {X 0,Y 591.089,Z 972.294,A -85,B 0,C 180,E1 27478.492,E2 27478.492} C_VEL
LIN {X 0,Y 588.706,Z 992.248,A -85,B 0,C 180,E1 27477.077,E2 27477.077} C_VEL
LIN {X 0,Y 586.509,Z 1010.193,A -85,B 0,C 180,E1 27475.597,E2 27475.597} C_VEL
LIN {X 0,Y 584.374,Z 1026.961,A -85,B 0,C 180,E1 27473.978,E2 27473.978} C_VEL
LIN {X 0,Y 582.386,Z 1043.11,A -85,B 0,C 180,E1 27472.192,E2 27472.192} C_VEL
LIN {X 0,Y 580.591,Z 1058.111,A -85,B 0,C 180,E1 27470.253,E2 27470.253} C_VEL
LIN {X 0,Y 579.06,Z 1072.41,A -85,B 0,C 180,E1 27468.108,E2 27468.108} C_VEL
LIN {X 0,Y 577.963,Z 1084.095,A -85,B 0,C 180,E1 27466.07,E2 27466.07} C_VEL
LIN {X 0,Y 577.122,Z 1094.429,A -85,B 0,C 180,E1 27463.935,E2 27463.935} C_VEL
LIN {X 0,Y 576.553,Z 1103.544,A -85,B 0,C 180,E1 27461.707,E2 27461.707} C_VEL
LIN {X 0,Y 576.204,Z 1110.778,A -85,B 0,C 180,E1 27459.489,E2 27459.489} C_VEL
LIN {X 0,Y 576.011,Z 1116.747,A -85,B 0,C 180,E1 27457.18,E2 27457.18} C_VEL
LIN {X 0,Y 575.928,Z 1120.791,A -85,B 0,C 180,E1 27454.98,E2 27454.98} C_VEL
LIN {X 0,Y 575.9,Z 1123.57,A -85,B 0,C 180,E1 27452.587,E2 27452.587} C_VEL
LIN {X 0,Y 575.899,Z 1124.55,A -85,B 0,C 180,E1 27450.497,E2 27450.497} C_VEL
LIN {X 0,Y 575.904,Z 1124.1,A -85,B 0,C 180,E1 27448.11,E2 27448.11} C_VEL
LIN {X 0,Y 575.914,Z 1122.263,A -85,B 0,C 180,E1 27446.018,E2 27446.018} C_VEL
LIN {X 0,Y 575.972,Z 1118.55,A -85,B 0,C 180,E1 27443.621,E2 27443.621} C_VEL
LIN {X 0,Y 576.098,Z 1113.811,A -85,B 0,C 180,E1 27441.516,E2 27441.516} C_VEL
LIN {X 0,Y 576.381,Z 1106.624,A -85,B 0,C 180,E1 27439.1,E2 27439.1} C_VEL
LIN {X 0,Y 576.847,Z 1098.635,A -85,B 0,C 180,E1 27436.947,E2 27436.947} C_VEL
LIN {X 0,Y 577.564,Z 1088.641,A -85,B 0,C 180,E1 27434.743,E2 27434.743} C_VEL
LIN {X 0,Y 578.589,Z 1077.269,A -85,B 0,C 180,E1 27432.604,E2 27432.604} C_VEL
LIN {X 0,Y 579.891,Z 1064.416,A -85,B 0,C 180,E1 27430.562,E2 27430.562} C_VEL
LIN {X 0,Y 581.667,Z 1048.847,A -85,B 0,C 180,E1 27428.433,E2 27428.433} C_VEL
LIN {X 0,Y 583.498,Z 1034.041,A -85,B 0,C 180,E1 27426.681,E2 27426.681} C_VEL
LIN {X 0,Y 585.556,Z 1017.57,A -85,B 0,C 180,E1 27424.999,E2 27424.999} C_VEL
LIN {X 0,Y 587.706,Z 1000.674,A -85,B 0,C 180,E1 27423.497,E2 27423.497} C_VEL
LIN {X 0,Y 589.971,Z 981.688,A -85,B 0,C 180,E1 27422.055,E2 27422.055} C_VEL
LIN {X 0,Y 592.236,Z 962.421,A -85,B 0,C 180,E1 27420.794,E2 27420.794} C_VEL
LIN {X 0,Y 594.324,Z 942.209,A -85,B 0,C 180,E1 27419.687,E2 27419.687} C_VEL
LIN {X 0,Y 596.34,Z 921.302,A -85,B 0,C 180,E1 27418.721,E2 27418.721} C_VEL
LIN {X 0,Y 598.009,Z 900.19,A -85,B 0,C 180,E1 27417.932,E2 27417.932} C_VEL
LIN {X 0,Y 599.596,Z 876.995,A -85,B 0,C 180,E1 27417.249,E2 27417.249} C_VEL
LIN {X 0,Y 600.62,Z 856.289,A -85,B 0,C 180,E1 27416.797,E2 27416.797} C_VEL
LIN {X 0,Y 601.412,Z 829.587,A -85,B 0,C 180,E1 27416.394,E2 27416.394} C_VEL
LIN {X 0,Y 605.833,Z 577.599,A -85,B 0,C 180,E1 27413.188,E2 27413.188} C_VEL
LIN {X 0,Y 606.511,Z 533.999,A -85,B 0,C 180,E1 27412.61,E2 27412.61} C_VEL
LIN {X 0,Y 598.138,Z 493.853,A -85,B 0,C 180,E1 27411.322,E2 27411.322} C_VEL
LIN {X 0,Y 599.227,Z 480.395,A -85,B 0,C 180,E1 27410.219,E2 27410.219} C_VEL
LIN {X 0,Y 592.61,Z 462.365,A -85,B 0,C 180,E1 27408.009,E2 27408.009} C_VEL
LIN {X 0,Y 585.064,Z 443.741,A -85,B 0,C 180,E1 27405.516,E2 27405.516} C_VEL
LIN {X 0,Y 580.065,Z 432.337,A -85,B 0,C 180,E1 27403.864,E2 27403.864} C_VEL
LIN {X 0,Y 577.331,Z 425.487,A -85,B 0,C 180,E1 27402.817,E2 27402.817} C_VEL
LIN {X 0,Y 577.227,Z 425.297,A -85,B 0,C 180,E1 27399.861,E2 27399.861} C_VEL
LIN {X 0,Y 577.295,Z 425.272,A -85,B 0,C 180,E1 27396.819,E2 27396.819} C_VEL
LIN {X 0,Y 577.225,Z 425.326,A -85,B 0,C 180,E1 27393.664,E2 27393.664} C_VEL
LIN {X 0,Y 577.283,Z 425.317,A -85,B 0,C 180,E1 27390.497,E2 27390.497} C_VEL
LIN {X 0,Y 577.219,Z 425.32,A -85,B 0,C 180,E1 27387.438,E2 27387.438} C_VEL
LIN {X 0,Y 577.26,Z 425.312,A -85,B 0,C 180,E1 27384.237,E2 27384.237} C_VEL
LIN {X 0,Y 577.225,Z 425.317,A -85,B 0,C 180,E1 27381.332,E2 27381.332} C_VEL
LIN {X 0,Y 577.261,Z 425.318,A -85,B 0,C 180,E1 27378.062,E2 27378.062} C_VEL
LIN {X 0,Y 577.241,Z 425.324,A -85,B 0,C 180,E1 27375.06,E2 27375.06} C_VEL
LIN {X 0,Y 577.246,Z 425.317,A -85,B 0,C 180,E1 27371.693,E2 27371.693} C_VEL
LIN {X 0,Y 577.262,Z 425.311,A -85,B 0,C 180,E1 27368.768,E2 27368.768} C_VEL
LIN {X 0,Y 577.252,Z 425.321,A -85,B 0,C 180,E1 27365.567,E2 27365.567} C_VEL
LIN {X 0,Y 577.288,Z 425.31,A -85,B 0,C 180,E1 27362.482,E2 27362.482} C_VEL
LIN {X 0,Y 577.25,Z 425.304,A -85,B 0,C 180,E1 27359.305,E2 27359.305} C_VEL
LIN {X 0,Y 577.311,Z 425.315,A -85,B 0,C 180,E1 27356.226,E2 27356.226} C_VEL
LIN {X 0,Y 577.257,Z 425.319,A -85,B 0,C 180,E1 27353.036,E2 27353.036} C_VEL
LIN {X 0,Y 577.313,Z 425.302,A -85,B 0,C 180,E1 27349.825,E2 27349.825} C_VEL
LIN {X 0,Y 577.268,Z 425.314,A -85,B 0,C 180,E1 27346.681,E2 27346.681} C_VEL
LIN {X 0,Y 577.291,Z 425.316,A -85,B 0,C 180,E1 27343.394,E2 27343.394} C_VEL
LIN {X 0,Y 577.3,Z 425.315,A -85,B 0,C 180,E1 27340.261,E2 27340.261} C_VEL
LIN {X 0,Y 577.278,Z 425.314,A -85,B 0,C 180,E1 27336.955,E2 27336.955} C_VEL
LIN {X 0,Y 577.321,Z 425.305,A -85,B 0,C 180,E1 27333.787,E2 27333.787} C_VEL
LIN {X 0,Y 577.278,Z 425.308,A -85,B 0,C 180,E1 27330.603,E2 27330.603} C_VEL
LIN {X 0,Y 577.318,Z 425.282,A -85,B 0,C 180,E1 27327.409,E2 27327.409} C_VEL
LIN {X 0,Y 577.297,Z 425.305,A -85,B 0,C 180,E1 27324.154,E2 27324.154} C_VEL
LIN {X 0,Y 577.289,Z 425.269,A -85,B 0,C 180,E1 27320.787,E2 27320.787} C_VEL
LIN {X 0,Y 577.342,Z 425.535,A -85,B 0,C 180,E1 27317.952,E2 27317.952} C_VEL
LIN {X 0,Y 578.95,Z 429.273,A -85,B 0,C 180,E1 27317.37,E2 27317.37} C_VEL
LIN {X 0,Y 587.526,Z 448.789,A -85,B 0,C 180,E1 27314.652,E2 27314.652} C_VEL
LIN {X 0,Y 591.566,Z 458.322,A -85,B 0,C 180,E1 27313.451,E2 27313.451} C_VEL
LIN {X 0,Y 606.802,Z 483.228,A -85,B 0,C 180,E1 27311.786,E2 27311.786} C_VEL
LIN {X 0,Y 609.024,Z 487.49,A -85,B 0,C 180,E1 27311.546,E2 27311.546} C_VEL
LIN {X 0,Y 609.8,Z 492.601,A -85,B 0,C 180,E1 27311.406,E2 27311.406} C_VEL
LIN {X 0,Y 604.159,Z 742.124,A -85,B 0,C 180,E1 27308.025,E2 27308.025} C_VEL
LIN {X 0,Y 601.87,Z 843.711,A -85,B 0,C 180,E1 27306.637,E2 27306.637} C_VEL
LIN {X 0,Y 600.672,Z 868.991,A -85,B 0,C 180,E1 27306.13,E2 27306.13} C_VEL
LIN {X 0,Y 599.372,Z 889.989,A -85,B 0,C 180,E1 27305.57,E2 27305.57} C_VEL
LIN {X 0,Y 597.589,Z 914.582,A -85,B 0,C 180,E1 27304.737,E2 27304.737} C_VEL
LIN {X 0,Y 595.781,Z 935.639,A -85,B 0,C 180,E1 27303.862,E2 27303.862} C_VEL
LIN {X 0,Y 593.752,Z 957.693,A -85,B 0,C 180,E1 27302.78,E2 27302.78} C_VEL
LIN {X 0,Y 591.591,Z 978.963,A -85,B 0,C 180,E1 27301.541,E2 27301.541} C_VEL
LIN {X 0,Y 589.332,Z 1000.698,A -85,B 0,C 180,E1 27300.083,E2 27300.083} C_VEL
LIN {X 0,Y 587.284,Z 1019.242,A -85,B 0,C 180,E1 27298.64,E2 27298.64} C_VEL
LIN {X 0,Y 585.239,Z 1038.132,A -85,B 0,C 180,E1 27296.976,E2 27296.976} C_VEL
LIN {X 0,Y 583.32,Z 1055.387,A -85,B 0,C 180,E1 27295.212,E2 27295.212} C_VEL
LIN {X 0,Y 581.639,Z 1071.433,A -85,B 0,C 180,E1 27293.365,E2 27293.365} C_VEL
LIN {X 0,Y 580.158,Z 1085.963,A -85,B 0,C 180,E1 27291.431,E2 27291.431} C_VEL
LIN {X 0,Y 578.991,Z 1098.281,A -85,B 0,C 180,E1 27289.574,E2 27289.574} C_VEL
LIN {X 0,Y 577.863,Z 1111.834,A -85,B 0,C 180,E1 27287.211,E2 27287.211} C_VEL
LIN {X 0,Y 577.167,Z 1121.6,A -85,B 0,C 180,E1 27285.213,E2 27285.213} C_VEL
LIN {X 0,Y 576.604,Z 1131.128,A -85,B 0,C 180,E1 27282.926,E2 27282.926} C_VEL
LIN {X 0,Y 576.246,Z 1138.512,A -85,B 0,C 180,E1 27280.7,E2 27280.7} C_VEL
LIN {X 0,Y 576.047,Z 1144.762,A -85,B 0,C 180,E1 27278.384,E2 27278.384} C_VEL
LIN {X 0,Y 575.948,Z 1149.493,A -85,B 0,C 180,E1 27275.979,E2 27275.979} C_VEL
LIN {X 0,Y 575.917,Z 1152.348,A -85,B 0,C 180,E1 27273.883,E2 27273.883} C_VEL
LIN {X 0,Y 575.901,Z 1154.189,A -85,B 0,C 180,E1 27271.393,E2 27271.393} C_VEL
LIN {X 0,Y 575.886,Z 1154.348,A -85,B 0,C 180,E1 27269.304,E2 27269.304} C_VEL
LIN {X 0,Y 575.889,Z 1153.425,A -85,B 0,C 180,E1 27267.313,E2 27267.313} C_VEL
LIN {X 0,Y 575.905,Z 1150.929,A -85,B 0,C 180,E1 27264.92,E2 27264.92} C_VEL
LIN {X 0,Y 575.97,Z 1147.101,A -85,B 0,C 180,E1 27262.719,E2 27262.719} C_VEL
LIN {X 0,Y 576.095,Z 1142.474,A -85,B 0,C 180,E1 27260.711,E2 27260.711} C_VEL
LIN {X 0,Y 576.371,Z 1135.364,A -85,B 0,C 180,E1 27258.289,E2 27258.289} C_VEL
LIN {X 0,Y 576.76,Z 1127.909,A -85,B 0,C 180,E1 27256.26,E2 27256.26} C_VEL
LIN {X 0,Y 577.341,Z 1119.015,A -85,B 0,C 180,E1 27254.222,E2 27254.222} C_VEL
LIN {X 0,Y 578.268,Z 1106.821,A -85,B 0,C 180,E1 27251.866,E2 27251.866} C_VEL
LIN {X 0,Y 579.32,Z 1094.812,A -85,B 0,C 180,E1 27249.873,E2 27249.873} C_VEL
LIN {X 0,Y 580.822,Z 1079.199,A -85,B 0,C 180,E1 27247.638,E2 27247.638} C_VEL
LIN {X 0,Y 582.293,Z 1065.076,A -85,B 0,C 180,E1 27245.878,E2 27245.878} C_VEL
LIN {X 0,Y 584.293,Z 1046.52,A -85,B 0,C 180,E1 27243.854,E2 27243.854} C_VEL
LIN {X 0,Y 586.167,Z 1029.562,A -85,B 0,C 180,E1 27242.245,E2 27242.245} C_VEL
LIN {X 0,Y 588.491,Z 1008.199,A -85,B 0,C 180,E1 27240.48,E2 27240.48} C_VEL
LIN {X 0,Y 590.503,Z 989.378,A -85,B 0,C 180,E1 27239.132,E2 27239.132} C_VEL
LIN {X 0,Y 592.844,Z 966.902,A -85,B 0,C 180,E1 27237.737,E2 27237.737} C_VEL
LIN {X 0,Y 594.749,Z 946.976,A -85,B 0,C 180,E1 27236.674,E2 27236.674} C_VEL
LIN {X 0,Y 596.817,Z 923.822,A -85,B 0,C 180,E1 27235.625,E2 27235.625} C_VEL
LIN {X 0,Y 598.514,Z 901.768,A -85,B 0,C 180,E1 27234.805,E2 27234.805} C_VEL
LIN {X 0,Y 600.207,Z 877.255,A -85,B 0,C 180,E1 27234.071,E2 27234.071} C_VEL
LIN {X 0,Y 601.393,Z 855.132,A -85,B 0,C 180,E1 27233.574,E2 27233.574} C_VEL
LIN {X 0,Y 602.289,Z 830.664,A -85,B 0,C 180,E1 27233.166,E2 27233.166} C_VEL
LIN {X 0,Y 607.47,Z 591.328,A -85,B 0,C 180,E1 27229.933,E2 27229.933} C_VEL
LIN {X 0,Y 609.651,Z 490.679,A -85,B 0,C 180,E1 27228.555,E2 27228.555} C_VEL
LIN {X 0,Y 608.571,Z 486.275,A -85,B 0,C 180,E1 27228.403,E2 27228.403} C_VEL
LIN {X 0,Y 593.625,Z 461.668,A -85,B 0,C 180,E1 27226.796,E2 27226.796} C_VEL
LIN {X 0,Y 591.275,Z 457.796,A -85,B 0,C 180,E1 27226.507,E2 27226.507} C_VEL
LIN {X 0,Y 583.792,Z 440.254,A -85,B 0,C 180,E1 27224.194,E2 27224.194} C_VEL
LIN {X 0,Y 578.477,Z 428.559,A -85,B 0,C 180,E1 27222.52,E2 27222.52} C_VEL
LIN {X 0,Y 577.34,Z 425.514,A -85,B 0,C 180,E1 27222.049,E2 27222.049} C_VEL
LIN {X 0,Y 577.32,Z 425.268,A -85,B 0,C 180,E1 27218.796,E2 27218.796} C_VEL
LIN {X 0,Y 577.284,Z 425.294,A -85,B 0,C 180,E1 27215.504,E2 27215.504} C_VEL
LIN {X 0,Y 577.317,Z 425.293,A -85,B 0,C 180,E1 27212.239,E2 27212.239} C_VEL
LIN {X 0,Y 577.284,Z 425.307,A -85,B 0,C 180,E1 27209.125,E2 27209.125} C_VEL
LIN {X 0,Y 577.308,Z 425.305,A -85,B 0,C 180,E1 27205.878,E2 27205.878} C_VEL
LIN {X 0,Y 577.296,Z 425.308,A -85,B 0,C 180,E1 27202.721,E2 27202.721} C_VEL
LIN {X 0,Y 577.278,Z 425.313,A -85,B 0,C 180,E1 27199.424,E2 27199.424} C_VEL
LIN {X 0,Y 577.323,Z 425.316,A -85,B 0,C 180,E1 27196.191,E2 27196.191} C_VEL
LIN {X 0,Y 577.265,Z 425.319,A -85,B 0,C 180,E1 27193.115,E2 27193.115} C_VEL
LIN {X 0,Y 577.32,Z 425.301,A -85,B 0,C 180,E1 27189.974,E2 27189.974} C_VEL
LIN {X 0,Y 577.261,Z 425.319,A -85,B 0,C 180,E1 27186.864,E2 27186.864} C_VEL
LIN {X 0,Y 577.307,Z 425.317,A -85,B 0,C 180,E1 27183.674,E2 27183.674} C_VEL
LIN {X 0,Y 577.256,Z 425.304,A -85,B 0,C 180,E1 27180.595,E2 27180.595} C_VEL
LIN {X 0,Y 577.272,Z 425.309,A -85,B 0,C 180,E1 27177.289,E2 27177.289} C_VEL
LIN {X 0,Y 577.269,Z 425.32,A -85,B 0,C 180,E1 27174.234,E2 27174.234} C_VEL
LIN {X 0,Y 577.248,Z 425.317,A -85,B 0,C 180,E1 27170.931,E2 27170.931} C_VEL
LIN {X 0,Y 577.285,Z 425.308,A -85,B 0,C 180,E1 27167.902,E2 27167.902} C_VEL
LIN {X 0,Y 577.239,Z 425.323,A -85,B 0,C 180,E1 27164.734,E2 27164.734} C_VEL
LIN {X 0,Y 577.299,Z 425.316,A -85,B 0,C 180,E1 27161.625,E2 27161.625} C_VEL
LIN {X 0,Y 577.228,Z 425.318,A -85,B 0,C 180,E1 27158.455,E2 27158.455} C_VEL
LIN {X 0,Y 577.299,Z 425.306,A -85,B 0,C 180,E1 27155.411,E2 27155.411} C_VEL
LIN {X 0,Y 577.224,Z 425.318,A -85,B 0,C 180,E1 27152.274,E2 27152.274} C_VEL
LIN {X 0,Y 577.283,Z 425.312,A -85,B 0,C 180,E1 27149.157,E2 27149.157} C_VEL
LIN {X 0,Y 577.219,Z 425.319,A -85,B 0,C 180,E1 27146.073,E2 27146.073} C_VEL
LIN {X 0,Y 577.249,Z 425.284,A -85,B 0,C 180,E1 27142.805,E2 27142.805} C_VEL
LIN {X 0,Y 577.221,Z 425.295,A -85,B 0,C 180,E1 27139.966,E2 27139.966} C_VEL
LIN {X 0,Y 577.328,Z 425.522,A -85,B 0,C 180,E1 27137.067,E2 27137.067} C_VEL
LIN {X 0,Y 580.158,Z 432.512,A -85,B 0,C 180,E1 27136.007,E2 27136.007} C_VEL
LIN {X 0,Y 585.663,Z 445.15,A -85,B 0,C 180,E1 27134.188,E2 27134.188} C_VEL
LIN {X 0,Y 593.194,Z 463.98,A -85,B 0,C 180,E1 27131.692,E2 27131.692} C_VEL
LIN {X 0,Y 599.289,Z 480.591,A -85,B 0,C 180,E1 27129.663,E2 27129.663} C_VEL
LIN {X 0,Y 598.182,Z 494.757,A -85,B 0,C 180,E1 27128.538,E2 27128.538} C_VEL
LIN {X 0,Y 606.665,Z 535.501,A -85,B 0,C 180,E1 27127.263,E2 27127.263} C_VEL
LIN {X 0,Y 605.065,Z 616.995,A -85,B 0,C 180,E1 27126.217,E2 27126.217} C_VEL
LIN {X 0,Y 604.158,Z 624.694,A -85,B 0,C 180,E1 27126.175,E2 27126.175} C_VEL
LIN {X 0,Y 598.83,Z 645.24,A -85,B 0,C 180,E1 27126.281,E2 27126.281} C_VEL
LIN {X 0,Y 598.122,Z 651.848,A -85,B 0,C 180,E1 27126.239,E2 27126.239} C_VEL
LIN {X 0,Y 594.447,Z 846.877,A -85,B 0,C 180,E1 27123.723,E2 27123.723} C_VEL
LIN {X 0,Y 593.355,Z 870.602,A -85,B 0,C 180,E1 27123.258,E2 27123.258} C_VEL
LIN {X 0,Y 592.035,Z 891.749,A -85,B 0,C 180,E1 27122.689,E2 27122.689} C_VEL
LIN {X 0,Y 590.23,Z 914.12,A -85,B 0,C 180,E1 27121.908,E2 27121.908} C_VEL
LIN {X 0,Y 588.245,Z 935.246,A -85,B 0,C 180,E1 27121,E2 27121} C_VEL
LIN {X 0,Y 586.005,Z 955.911,A -85,B 0,C 180,E1 27119.911,E2 27119.911} C_VEL
LIN {X 0,Y 583.688,Z 976.044,A -85,B 0,C 180,E1 27118.663,E2 27118.663} C_VEL
LIN {X 0,Y 581.315,Z 994.578,A -85,B 0,C 180,E1 27117.301,E2 27117.301} C_VEL
LIN {X 0,Y 578.924,Z 1013.098,A -85,B 0,C 180,E1 27115.727,E2 27115.727} C_VEL
LIN {X 0,Y 576.8,Z 1029.046,A -85,B 0,C 180,E1 27114.149,E2 27114.149} C_VEL
LIN {X 0,Y 574.593,Z 1045.951,A -85,B 0,C 180,E1 27112.214,E2 27112.214} C_VEL
LIN {X 0,Y 572.875,Z 1059.62,A -85,B 0,C 180,E1 27110.4,E2 27110.4} C_VEL
LIN {X 0,Y 571.274,Z 1073.504,A -85,B 0,C 180,E1 27108.258,E2 27108.258} C_VEL
LIN {X 0,Y 570.064,Z 1085.59,A -85,B 0,C 180,E1 27106.089,E2 27106.089} C_VEL
LIN {X 0,Y 569.179,Z 1095.669,A -85,B 0,C 180,E1 27103.926,E2 27103.926} C_VEL
LIN {X 0,Y 568.553,Z 1104.891,A -85,B 0,C 180,E1 27101.566,E2 27101.566} C_VEL
LIN {X 0,Y 568.215,Z 1111.647,A -85,B 0,C 180,E1 27099.419,E2 27099.419} C_VEL
LIN {X 0,Y 568,Z 1117.596,A -85,B 0,C 180,E1 27096.977,E2 27096.977} C_VEL
LIN {X 0,Y 567.928,Z 1121.328,A -85,B 0,C 180,E1 27094.848,E2 27094.848} C_VEL
LIN {X 0,Y 567.905,Z 1123.918,A -85,B 0,C 180,E1 27092.422,E2 27092.422} C_VEL
LIN {X 0,Y 567.909,Z 1124.829,A -85,B 0,C 180,E1 27090.202,E2 27090.202} C_VEL
LIN {X 0,Y 567.909,Z 1124.178,A -85,B 0,C 180,E1 27087.881,E2 27087.881} C_VEL
LIN {X 0,Y 567.923,Z 1122.259,A -85,B 0,C 180,E1 27085.759,E2 27085.759} C_VEL
LIN {X 0,Y 567.981,Z 1118.583,A -85,B 0,C 180,E1 27083.429,E2 27083.429} C_VEL
LIN {X 0,Y 568.125,Z 1113.815,A -85,B 0,C 180,E1 27081.294,E2 27081.294} C_VEL
LIN {X 0,Y 568.437,Z 1106.913,A -85,B 0,C 180,E1 27078.946,E2 27078.946} C_VEL
LIN {X 0,Y 568.939,Z 1099.075,A -85,B 0,C 180,E1 27076.793,E2 27076.793} C_VEL
LIN {X 0,Y 569.727,Z 1089.017,A -85,B 0,C 180,E1 27074.528,E2 27074.528} C_VEL
LIN {X 0,Y 570.844,Z 1077.601,A -85,B 0,C 180,E1 27072.34,E2 27072.34} C_VEL
LIN {X 0,Y 572.238,Z 1064.922,A -85,B 0,C 180,E1 27070.291,E2 27070.291} C_VEL
LIN {X 0,Y 574.105,Z 1049.727,A -85,B 0,C 180,E1 27068.172,E2 27068.172} C_VEL
LIN {X 0,Y 575.986,Z 1035.252,A -85,B 0,C 180,E1 27066.433,E2 27066.433} C_VEL
LIN {X 0,Y 578.241,Z 1018.139,A -85,B 0,C 180,E1 27064.661,E2 27064.661} C_VEL
LIN {X 0,Y 580.452,Z 1001.505,A -85,B 0,C 180,E1 27063.166,E2 27063.166} C_VEL
LIN {X 0,Y 582.786,Z 982.992,A -85,B 0,C 180,E1 27061.736,E2 27061.736} C_VEL
LIN {X 0,Y 585.141,Z 963.858,A -85,B 0,C 180,E1 27060.463,E2 27060.463} C_VEL
LIN {X 0,Y 587.331,Z 943.885,A -85,B 0,C 180,E1 27059.344,E2 27059.344} C_VEL
LIN {X 0,Y 589.402,Z 923.633,A -85,B 0,C 180,E1 27058.385,E2 27058.385} C_VEL
LIN {X 0,Y 591.205,Z 902.164,A -85,B 0,C 180,E1 27057.56,E2 27057.56} C_VEL
LIN {X 0,Y 592.882,Z 879.532,A -85,B 0,C 180,E1 27056.867,E2 27056.867} C_VEL
LIN {X 0,Y 594.031,Z 857.485,A -85,B 0,C 180,E1 27056.373,E2 27056.373} C_VEL
LIN {X 0,Y 594.846,Z 833.501,A -85,B 0,C 180,E1 27055.994,E2 27055.994} C_VEL
LIN {X 0,Y 599.461,Z 583.901,A -85,B 0,C 180,E1 27052.791,E2 27052.791} C_VEL
LIN {X 0,Y 600.309,Z 535.718,A -85,B 0,C 180,E1 27052.151,E2 27052.151} C_VEL
LIN {X 0,Y 591.553,Z 493.57,A -85,B 0,C 180,E1 27050.774,E2 27050.774} C_VEL
LIN {X 0,Y 592.38,Z 483.91,A -85,B 0,C 180,E1 27049.977,E2 27049.977} C_VEL
LIN {X 0,Y 585.639,Z 465.379,A -85,B 0,C 180,E1 27047.671,E2 27047.671} C_VEL
LIN {X 0,Y 578.465,Z 447.789,A -85,B 0,C 180,E1 27045.27,E2 27045.27} C_VEL
LIN {X 0,Y 573.661,Z 436.761,A -85,B 0,C 180,E1 27043.648,E2 27043.648} C_VEL
LIN {X 0,Y 570.574,Z 429.676,A -85,B 0,C 180,E1 27042.566,E2 27042.566} C_VEL
LIN {X 0,Y 569.319,Z 426.462,A -85,B 0,C 180,E1 27042.02,E2 27042.02} C_VEL
LIN {X 0,Y 569.309,Z 426.298,A -85,B 0,C 180,E1 27039.349,E2 27039.349} C_VEL
LIN {X 0,Y 569.29,Z 426.259,A -85,B 0,C 180,E1 27036.043,E2 27036.043} C_VEL
LIN {X 0,Y 569.331,Z 426.315,A -85,B 0,C 180,E1 27032.987,E2 27032.987} C_VEL
LIN {X 0,Y 569.284,Z 426.318,A -85,B 0,C 180,E1 27029.806,E2 27029.806} C_VEL
LIN {X 0,Y 569.345,Z 426.31,A -85,B 0,C 180,E1 27026.718,E2 27026.718} C_VEL
LIN {X 0,Y 569.283,Z 426.313,A -85,B 0,C 180,E1 27023.497,E2 27023.497} C_VEL
LIN {X 0,Y 569.348,Z 426.296,A -85,B 0,C 180,E1 27020.349,E2 27020.349} C_VEL
LIN {X 0,Y 569.292,Z 426.303,A -85,B 0,C 180,E1 27017.267,E2 27017.267} C_VEL
LIN {X 0,Y 569.331,Z 426.307,A -85,B 0,C 180,E1 27014.026,E2 27014.026} C_VEL
LIN {X 0,Y 569.305,Z 426.309,A -85,B 0,C 180,E1 27011.037,E2 27011.037} C_VEL
LIN {X 0,Y 569.313,Z 426.298,A -85,B 0,C 180,E1 27007.671,E2 27007.671} C_VEL
LIN {X 0,Y 569.327,Z 426.303,A -85,B 0,C 180,E1 27004.735,E2 27004.735} C_VEL
LIN {X 0,Y 569.313,Z 426.312,A -85,B 0,C 180,E1 27001.409,E2 27001.409} C_VEL
LIN {X 0,Y 569.357,Z 426.292,A -85,B 0,C 180,E1 26998.39,E2 26998.39} C_VEL
LIN {X 0,Y 569.315,Z 426.299,A -85,B 0,C 180,E1 26995.164,E2 26995.164} C_VEL
LIN {X 0,Y 569.387,Z 426.304,A -85,B 0,C 180,E1 26992.026,E2 26992.026} C_VEL
LIN {X 0,Y 569.327,Z 426.305,A -85,B 0,C 180,E1 26988.758,E2 26988.758} C_VEL
LIN {X 0,Y 569.346,Z 426.294,A -85,B 0,C 180,E1 26985.393,E2 26985.393} C_VEL
LIN {X 0,Y 569.354,Z 426.295,A -85,B 0,C 180,E1 26982.313,E2 26982.313} C_VEL
LIN {X 0,Y 569.337,Z 426.306,A -85,B 0,C 180,E1 26979.006,E2 26979.006} C_VEL
LIN {X 0,Y 569.384,Z 426.306,A -85,B 0,C 180,E1 26975.847,E2 26975.847} C_VEL
LIN {X 0,Y 569.342,Z 426.31,A -85,B 0,C 180,E1 26972.604,E2 26972.604} C_VEL
LIN {X 0,Y 569.383,Z 426.307,A -85,B 0,C 180,E1 26969.372,E2 26969.372} C_VEL
LIN {X 0,Y 569.362,Z 426.251,A -85,B 0,C 180,E1 26966.051,E2 26966.051} C_VEL
LIN {X 0,Y 569.351,Z 426.3,A -85,B 0,C 180,E1 26962.707,E2 26962.707} C_VEL
LIN {X 0,Y 569.375,Z 426.267,A -85,B 0,C 180,E1 26959.476,E2 26959.476} C_VEL
LIN {X 0,Y 569.412,Z 426.683,A -85,B 0,C 180,E1 26958.694,E2 26958.694} C_VEL
LIN {X 0,Y 570.934,Z 430.186,A -85,B 0,C 180,E1 26958.144,E2 26958.144} C_VEL
LIN {X 0,Y 578.473,Z 447.074,A -85,B 0,C 180,E1 26955.693,E2 26955.693} C_VEL
LIN {X 0,Y 583.53,Z 458.765,A -85,B 0,C 180,E1 26954.148,E2 26954.148} C_VEL
LIN {X 0,Y 597.694,Z 481.58,A -85,B 0,C 180,E1 26952.548,E2 26952.548} C_VEL
LIN {X 0,Y 603.284,Z 491.445,A -85,B 0,C 180,E1 26951.938,E2 26951.938} C_VEL
LIN {X 0,Y 603.58,Z 494.952,A -85,B 0,C 180,E1 26951.859,E2 26951.859} C_VEL
LIN {X 0,Y 597.665,Z 743.584,A -85,B 0,C 180,E1 26948.458,E2 26948.458} C_VEL
LIN {X 0,Y 595.283,Z 843.762,A -85,B 0,C 180,E1 26947.074,E2 26947.074} C_VEL
LIN {X 0,Y 594.026,Z 868.972,A -85,B 0,C 180,E1 26946.564,E2 26946.564} C_VEL
LIN {X 0,Y 592.649,Z 890.205,A -85,B 0,C 180,E1 26945.991,E2 26945.991} C_VEL
LIN {X 0,Y 590.735,Z 915.143,A -85,B 0,C 180,E1 26945.134,E2 26945.134} C_VEL
LIN {X 0,Y 588.878,Z 935.762,A -85,B 0,C 180,E1 26944.266,E2 26944.266} C_VEL
LIN {X 0,Y 586.72,Z 957.899,A -85,B 0,C 180,E1 26943.165,E2 26943.165} C_VEL
LIN {X 0,Y 584.494,Z 978.513,A -85,B 0,C 180,E1 26941.95,E2 26941.95} C_VEL
LIN {X 0,Y 582.175,Z 999.652,A -85,B 0,C 180,E1 26940.518,E2 26940.518} C_VEL
LIN {X 0,Y 579.889,Z 1019.124,A -85,B 0,C 180,E1 26938.981,E2 26938.981} C_VEL
LIN {X 0,Y 577.726,Z 1037.995,A -85,B 0,C 180,E1 26937.3,E2 26937.3} C_VEL
LIN {X 0,Y 575.72,Z 1055.263,A -85,B 0,C 180,E1 26935.513,E2 26935.513} C_VEL
LIN {X 0,Y 573.897,Z 1071.761,A -85,B 0,C 180,E1 26933.588,E2 26933.588} C_VEL
LIN {X 0,Y 572.346,Z 1086.197,A -85,B 0,C 180,E1 26931.631,E2 26931.631} C_VEL
LIN {X 0,Y 571.18,Z 1097.842,A -85,B 0,C 180,E1 26929.853,E2 26929.853} C_VEL
LIN {X 0,Y 570.035,Z 1110.924,A -85,B 0,C 180,E1 26927.56,E2 26927.56} C_VEL
LIN {X 0,Y 569.261,Z 1120.996,A -85,B 0,C 180,E1 26925.485,E2 26925.485} C_VEL
LIN {X 0,Y 568.67,Z 1130.476,A -85,B 0,C 180,E1 26923.213,E2 26923.213} C_VEL
LIN {X 0,Y 568.266,Z 1138.391,A -85,B 0,C 180,E1 26920.852,E2 26920.852} C_VEL
LIN {X 0,Y 568.051,Z 1144.506,A -85,B 0,C 180,E1 26918.605,E2 26918.605} C_VEL
LIN {X 0,Y 567.954,Z 1149.333,A -85,B 0,C 180,E1 26916.165,E2 26916.165} C_VEL
LIN {X 0,Y 567.92,Z 1152.234,A -85,B 0,C 180,E1 26914.038,E2 26914.038} C_VEL
LIN {X 0,Y 567.898,Z 1154.144,A -85,B 0,C 180,E1 26911.614,E2 26911.614} C_VEL
LIN {X 0,Y 567.886,Z 1154.348,A -85,B 0,C 180,E1 26909.294,E2 26909.294} C_VEL
LIN {X 0,Y 567.888,Z 1153.425,A -85,B 0,C 180,E1 26907.275,E2 26907.275} C_VEL
LIN {X 0,Y 567.905,Z 1150.929,A -85,B 0,C 180,E1 26904.848,E2 26904.848} C_VEL
LIN {X 0,Y 567.972,Z 1147.101,A -85,B 0,C 180,E1 26902.616,E2 26902.616} C_VEL
LIN {X 0,Y 568.103,Z 1142.696,A -85,B 0,C 180,E1 26900.681,E2 26900.681} C_VEL
LIN {X 0,Y 568.369,Z 1135.891,A -85,B 0,C 180,E1 26898.328,E2 26898.328} C_VEL
LIN {X 0,Y 568.81,Z 1127.592,A -85,B 0,C 180,E1 26896.065,E2 26896.065} C_VEL
LIN {X 0,Y 569.463,Z 1118.193,A -85,B 0,C 180,E1 26893.893,E2 26893.893} C_VEL
LIN {X 0,Y 570.408,Z 1106.417,A -85,B 0,C 180,E1 26891.607,E2 26891.607} C_VEL
LIN {X 0,Y 571.515,Z 1094.601,A -85,B 0,C 180,E1 26889.625,E2 26889.625} C_VEL
LIN {X 0,Y 573.132,Z 1078.686,A -85,B 0,C 180,E1 26887.321,E2 26887.321} C_VEL
LIN {X 0,Y 574.724,Z 1064.135,A -85,B 0,C 180,E1 26885.493,E2 26885.493} C_VEL
LIN {X 0,Y 576.806,Z 1045.86,A -85,B 0,C 180,E1 26883.489,E2 26883.489} C_VEL
LIN {X 0,Y 578.709,Z 1029.421,A -85,B 0,C 180,E1 26881.912,E2 26881.912} C_VEL
LIN {X 0,Y 581.147,Z 1008.151,A -85,B 0,C 180,E1 26880.13,E2 26880.13} C_VEL
LIN {X 0,Y 583.296,Z 989.41,A -85,B 0,C 180,E1 26878.765,E2 26878.765} C_VEL
LIN {X 0,Y 585.852,Z 966.154,A -85,B 0,C 180,E1 26877.304,E2 26877.304} C_VEL
LIN {X 0,Y 587.902,Z 945.778,A -85,B 0,C 180,E1 26876.21,E2 26876.21} C_VEL
LIN {X 0,Y 590.16,Z 921.625,A -85,B 0,C 180,E1 26875.123,E2 26875.123} C_VEL
LIN {X 0,Y 591.846,Z 900.796,A -85,B 0,C 180,E1 26874.348,E2 26874.348} C_VEL
LIN {X 0,Y 593.649,Z 875.36,A -85,B 0,C 180,E1 26873.594,E2 26873.594} C_VEL
LIN {X 0,Y 594.826,Z 854.286,A -85,B 0,C 180,E1 26873.122,E2 26873.122} C_VEL
LIN {X 0,Y 595.75,Z 829.21,A -85,B 0,C 180,E1 26872.707,E2 26872.707} C_VEL
LIN {X 0,Y 601.2,Z 590.718,A -85,B 0,C 180,E1 26869.452,E2 26869.452} C_VEL
LIN {X 0,Y 603.456,Z 492.412,A -85,B 0,C 180,E1 26868.095,E2 26868.095} C_VEL
LIN {X 0,Y 602.667,Z 490.027,A -85,B 0,C 180,E1 26867.994,E2 26867.994} C_VEL
LIN {X 0,Y 588.343,Z 466.422,A -85,B 0,C 180,E1 26866.42,E2 26866.42} C_VEL
LIN {X 0,Y 583.149,Z 458.028,A -85,B 0,C 180,E1 26865.785,E2 26865.785} C_VEL
LIN {X 0,Y 575.75,Z 440.971,A -85,B 0,C 180,E1 26863.45,E2 26863.45} C_VEL
LIN {X 0,Y 570.901,Z 430.138,A -85,B 0,C 180,E1 26861.859,E2 26861.859} C_VEL
LIN {X 0,Y 569.382,Z 426.487,A -85,B 0,C 180,E1 26861.27,E2 26861.27} C_VEL
LIN {X 0,Y 569.374,Z 426.269,A -85,B 0,C 180,E1 26858.117,E2 26858.117} C_VEL
LIN {X 0,Y 569.363,Z 426.261,A -85,B 0,C 180,E1 26854.902,E2 26854.902} C_VEL
LIN {X 0,Y 569.347,Z 426.302,A -85,B 0,C 180,E1 26851.557,E2 26851.557} C_VEL
LIN {X 0,Y 569.386,Z 426.297,A -85,B 0,C 180,E1 26848.304,E2 26848.304} C_VEL
LIN {X 0,Y 569.343,Z 426.303,A -85,B 0,C 180,E1 26845.04,E2 26845.04} C_VEL
LIN {X 0,Y 569.353,Z 426.296,A -85,B 0,C 180,E1 26841.642,E2 26841.642} C_VEL
LIN {X 0,Y 569.372,Z 426.289,A -85,B 0,C 180,E1 26838.428,E2 26838.428} C_VEL
LIN {X 0,Y 569.329,Z 426.301,A -85,B 0,C 180,E1 26835.17,E2 26835.17} C_VEL
LIN {X 0,Y 569.382,Z 426.308,A -85,B 0,C 180,E1 26831.96,E2 26831.96} C_VEL
LIN {X 0,Y 569.328,Z 426.305,A -85,B 0,C 180,E1 26828.789,E2 26828.789} C_VEL
LIN {X 0,Y 569.351,Z 426.291,A -85,B 0,C 180,E1 26825.543,E2 26825.543} C_VEL
LIN {X 0,Y 569.336,Z 426.309,A -85,B 0,C 180,E1 26822.416,E2 26822.416} C_VEL
LIN {X 0,Y 569.321,Z 426.313,A -85,B 0,C 180,E1 26819.094,E2 26819.094} C_VEL
LIN {X 0,Y 569.362,Z 426.288,A -85,B 0,C 180,E1 26815.951,E2 26815.951} C_VEL
LIN {X 0,Y 569.307,Z 426.303,A -85,B 0,C 180,E1 26812.837,E2 26812.837} C_VEL
LIN {X 0,Y 569.374,Z 426.308,A -85,B 0,C 180,E1 26809.681,E2 26809.681} C_VEL
LIN {X 0,Y 569.302,Z 426.307,A -85,B 0,C 180,E1 26806.491,E2 26806.491} C_VEL
LIN {X 0,Y 569.355,Z 426.293,A -85,B 0,C 180,E1 26803.366,E2 26803.366} C_VEL
LIN {X 0,Y 569.298,Z 426.312,A -85,B 0,C 180,E1 26800.29,E2 26800.29} C_VEL
LIN {X 0,Y 569.316,Z 426.312,A -85,B 0,C 180,E1 26796.971,E2 26796.971} C_VEL
LIN {X 0,Y 569.303,Z 426.312,A -85,B 0,C 180,E1 26793.954,E2 26793.954} C_VEL
LIN {X 0,Y 569.289,Z 426.318,A -85,B 0,C 180,E1 26790.595,E2 26790.595} C_VEL
LIN {X 0,Y 569.318,Z 426.306,A -85,B 0,C 180,E1 26787.61,E2 26787.61} C_VEL
LIN {X 0,Y 569.275,Z 426.263,A -85,B 0,C 180,E1 26784.413,E2 26784.413} C_VEL
LIN {X 0,Y 569.359,Z 426.313,A -85,B 0,C 180,E1 26781.237,E2 26781.237} C_VEL
LIN {X 0,Y 569.281,Z 426.269,A -85,B 0,C 180,E1 26778.13,E2 26778.13} C_VEL
LIN {X 0,Y 569.361,Z 426.735,A -85,B 0,C 180,E1 26777.799,E2 26777.799} C_VEL
LIN {X 0,Y 577.474,Z 445.275,A -85,B 0,C 180,E1 26774.983,E2 26774.983} C_VEL
LIN {X 0,Y 585.254,Z 464.396,A -85,B 0,C 180,E1 26772.361,E2 26772.361} C_VEL
LIN {X 0,Y 592.402,Z 484.004,A -85,B 0,C 180,E1 26769.917,E2 26769.917} C_VEL
LIN {X 0,Y 591.598,Z 494.394,A -85,B 0,C 180,E1 26769.089,E2 26769.089} C_VEL
LIN {X 0,Y 600.437,Z 537.123,A -85,B 0,C 180,E1 26767.725,E2 26767.725} C_VEL
LIN {X 0,Y 598.122,Z 651.848,A -85,B 0,C 180,E1 26766.239,E2 26766.239} C_VEL
LIN {X 0,Y 597.21,Z 659.547,A -85,B 0,C 180,E1 26766.198,E2 26766.198} C_VEL
LIN {X 0,Y 591.901,Z 680.096,A -85,B 0,C 180,E1 26766.304,E2 26766.304} C_VEL
LIN {X 0,Y 591.178,Z 686.705,A -85,B 0,C 180,E1 26766.264,E2 26766.264} C_VEL
LIN {X 0,Y 587.957,Z 847.022,A -85,B 0,C 180,E1 26764.178,E2 26764.178} C_VEL
LIN {X 0,Y 586.806,Z 870.778,A -85,B 0,C 180,E1 26763.708,E2 26763.708} C_VEL
LIN {X 0,Y 585.414,Z 892.132,A -85,B 0,C 180,E1 26763.128,E2 26763.128} C_VEL
LIN {X 0,Y 583.582,Z 913.912,A -85,B 0,C 180,E1 26762.361,E2 26762.361} C_VEL
LIN {X 0,Y 581.598,Z 934.12,A -85,B 0,C 180,E1 26761.49,E2 26761.49} C_VEL
LIN {X 0,Y 579.22,Z 955.188,A -85,B 0,C 180,E1 26760.384,E2 26760.384} C_VEL
LIN {X 0,Y 576.834,Z 975.091,A -85,B 0,C 180,E1 26759.15,E2 26759.15} C_VEL
LIN {X 0,Y 574.31,Z 993.996,A -85,B 0,C 180,E1 26757.757,E2 26757.757} C_VEL
LIN {X 0,Y 571.886,Z 1011.887,A -85,B 0,C 180,E1 26756.241,E2 26756.241} C_VEL
LIN {X 0,Y 569.533,Z 1028.662,A -85,B 0,C 180,E1 26754.574,E2 26754.574} C_VEL
LIN {X 0,Y 567.275,Z 1045.009,A -85,B 0,C 180,E1 26752.707,E2 26752.707} C_VEL
LIN {X 0,Y 565.392,Z 1059.179,A -85,B 0,C 180,E1 26750.822,E2 26750.822} C_VEL
LIN {X 0,Y 563.638,Z 1073.359,A -85,B 0,C 180,E1 26748.622,E2 26748.622} C_VEL
LIN {X 0,Y 562.307,Z 1085.487,A -85,B 0,C 180,E1 26746.423,E2 26746.423} C_VEL
LIN {X 0,Y 561.303,Z 1096.034,A -85,B 0,C 180,E1 26744.126,E2 26744.126} C_VEL
LIN {X 0,Y 560.622,Z 1105.243,A -85,B 0,C 180,E1 26741.716,E2 26741.716} C_VEL
LIN {X 0,Y 560.257,Z 1111.921,A -85,B 0,C 180,E1 26739.554,E2 26739.554} C_VEL
LIN {X 0,Y 560.021,Z 1117.843,A -85,B 0,C 180,E1 26737.077,E2 26737.077} C_VEL
LIN {X 0,Y 559.938,Z 1121.559,A -85,B 0,C 180,E1 26734.917,E2 26734.917} C_VEL
LIN {X 0,Y 559.909,Z 1124.133,A -85,B 0,C 180,E1 26732.456,E2 26732.456} C_VEL
LIN {X 0,Y 559.911,Z 1125.039,A -85,B 0,C 180,E1 26730.205,E2 26730.205} C_VEL
LIN {X 0,Y 559.911,Z 1124.391,A -85,B 0,C 180,E1 26727.851,E2 26727.851} C_VEL
LIN {X 0,Y 559.927,Z 1122.479,A -85,B 0,C 180,E1 26725.699,E2 26725.699} C_VEL
LIN {X 0,Y 559.993,Z 1118.822,A -85,B 0,C 180,E1 26723.335,E2 26723.335} C_VEL
LIN {X 0,Y 560.149,Z 1114.075,A -85,B 0,C 180,E1 26721.169,E2 26721.169} C_VEL
LIN {X 0,Y 560.495,Z 1107.209,A -85,B 0,C 180,E1 26718.787,E2 26718.787} C_VEL
LIN {X 0,Y 561.043,Z 1099.402,A -85,B 0,C 180,E1 26716.604,E2 26716.604} C_VEL
LIN {X 0,Y 561.904,Z 1089.377,A -85,B 0,C 180,E1 26714.301,E2 26714.301} C_VEL
LIN {X 0,Y 563.09,Z 1078.172,A -85,B 0,C 180,E1 26712.109,E2 26712.109} C_VEL
LIN {X 0,Y 564.594,Z 1065.425,A -85,B 0,C 180,E1 26710.013,E2 26710.013} C_VEL
LIN {X 0,Y 566.419,Z 1051.447,A -85,B 0,C 180,E1 26708.023,E2 26708.023} C_VEL
LIN {X 0,Y 568.385,Z 1036.906,A -85,B 0,C 180,E1 26706.243,E2 26706.243} C_VEL
LIN {X 0,Y 570.858,Z 1019.164,A -85,B 0,C 180,E1 26704.365,E2 26704.365} C_VEL
LIN {X 0,Y 573.07,Z 1003.243,A -85,B 0,C 180,E1 26702.91,E2 26702.91} C_VEL
LIN {X 0,Y 575.704,Z 983.525,A -85,B 0,C 180,E1 26701.356,E2 26701.356} C_VEL
LIN {X 0,Y 578.058,Z 965.209,A -85,B 0,C 180,E1 26700.121,E2 26700.121} C_VEL
LIN {X 0,Y 580.459,Z 944.524,A -85,B 0,C 180,E1 26698.941,E2 26698.941} C_VEL
LIN {X 0,Y 582.616,Z 924.326,A -85,B 0,C 180,E1 26697.974,E2 26697.974} C_VEL
LIN {X 0,Y 584.54,Z 902.655,A -85,B 0,C 180,E1 26697.128,E2 26697.128} C_VEL
LIN {X 0,Y 586.27,Z 880.361,A -85,B 0,C 180,E1 26696.437,E2 26696.437} C_VEL
LIN {X 0,Y 587.497,Z 858.137,A -85,B 0,C 180,E1 26695.93,E2 26695.93} C_VEL
LIN {X 0,Y 588.354,Z 834.768,A -85,B 0,C 180,E1 26695.552,E2 26695.552} C_VEL
LIN {X 0,Y 593.218,Z 585.661,A -85,B 0,C 180,E1 26692.326,E2 26692.326} C_VEL
LIN {X 0,Y 594.119,Z 537.356,A -85,B 0,C 180,E1 26691.678,E2 26691.678} C_VEL
LIN {X 0,Y 585.02,Z 493.119,A -85,B 0,C 180,E1 26690.202,E2 26690.202} C_VEL
LIN {X 0,Y 585.44,Z 487.061,A -85,B 0,C 180,E1 26689.686,E2 26689.686} C_VEL
LIN {X 0,Y 578.176,Z 467.2,A -85,B 0,C 180,E1 26687.161,E2 26687.161} C_VEL
LIN {X 0,Y 570.79,Z 449.094,A -85,B 0,C 180,E1 26684.625,E2 26684.625} C_VEL
LIN {X 0,Y 564.248,Z 434.304,A -85,B 0,C 180,E1 26682.357,E2 26682.357} C_VEL
LIN {X 0,Y 561.417,Z 427.493,A -85,B 0,C 180,E1 26681.237,E2 26681.237} C_VEL
LIN {X 0,Y 561.377,Z 427.3,A -85,B 0,C 180,E1 26678.304,E2 26678.304} C_VEL
LIN {X 0,Y 561.365,Z 427.249,A -85,B 0,C 180,E1 26675.247,E2 26675.247} C_VEL
LIN {X 0,Y 561.349,Z 427.294,A -85,B 0,C 180,E1 26671.94,E2 26671.94} C_VEL
LIN {X 0,Y 561.377,Z 427.296,A -85,B 0,C 180,E1 26668.978,E2 26668.978} C_VEL
LIN {X 0,Y 561.344,Z 427.303,A -85,B 0,C 180,E1 26665.761,E2 26665.761} C_VEL
LIN {X 0,Y 561.415,Z 427.302,A -85,B 0,C 180,E1 26662.625,E2 26662.625} C_VEL
LIN {X 0,Y 561.35,Z 427.302,A -85,B 0,C 180,E1 26659.456,E2 26659.456} C_VEL
LIN {X 0,Y 561.409,Z 427.284,A -85,B 0,C 180,E1 26656.238,E2 26656.238} C_VEL
LIN {X 0,Y 561.355,Z 427.294,A -85,B 0,C 180,E1 26653.284,E2 26653.284} C_VEL
LIN {X 0,Y 561.407,Z 427.297,A -85,B 0,C 180,E1 26650.052,E2 26650.052} C_VEL
LIN {X 0,Y 561.372,Z 427.292,A -85,B 0,C 180,E1 26646.957,E2 26646.957} C_VEL
LIN {X 0,Y 561.377,Z 427.28,A -85,B 0,C 180,E1 26643.574,E2 26643.574} C_VEL
LIN {X 0,Y 561.407,Z 427.293,A -85,B 0,C 180,E1 26640.51,E2 26640.51} C_VEL
LIN {X 0,Y 561.378,Z 427.3,A -85,B 0,C 180,E1 26637.244,E2 26637.244} C_VEL
LIN {X 0,Y 561.442,Z 427.279,A -85,B 0,C 180,E1 26633.968,E2 26633.968} C_VEL
LIN {X 0,Y 561.383,Z 427.29,A -85,B 0,C 180,E1 26630.879,E2 26630.879} C_VEL
LIN {X 0,Y 561.418,Z 427.294,A -85,B 0,C 180,E1 26627.555,E2 26627.555} C_VEL
LIN {X 0,Y 561.409,Z 427.292,A -85,B 0,C 180,E1 26624.399,E2 26624.399} C_VEL
LIN {X 0,Y 561.397,Z 427.286,A -85,B 0,C 180,E1 26621.042,E2 26621.042} C_VEL
LIN {X 0,Y 561.447,Z 427.277,A -85,B 0,C 180,E1 26617.818,E2 26617.818} C_VEL
LIN {X 0,Y 561.401,Z 427.286,A -85,B 0,C 180,E1 26614.556,E2 26614.556} C_VEL
LIN {X 0,Y 561.425,Z 427.283,A -85,B 0,C 180,E1 26611.193,E2 26611.193} C_VEL
LIN {X 0,Y 561.435,Z 427.273,A -85,B 0,C 180,E1 26607.945,E2 26607.945} C_VEL
LIN {X 0,Y 561.404,Z 427.262,A -85,B 0,C 180,E1 26604.631,E2 26604.631} C_VEL
LIN {X 0,Y 561.436,Z 427.246,A -85,B 0,C 180,E1 26601.43,E2 26601.43} C_VEL
LIN {X 0,Y 561.47,Z 427.501,A -85,B 0,C 180,E1 26599.544,E2 26599.544} C_VEL
LIN {X 0,Y 563.047,Z 431.235,A -85,B 0,C 180,E1 26598.923,E2 26598.923} C_VEL
LIN {X 0,Y 570.457,Z 447.563,A -85,B 0,C 180,E1 26596.461,E2 26596.461} C_VEL
LIN {X 0,Y 575.492,Z 459.206,A -85,B 0,C 180,E1 26594.873,E2 26594.873} C_VEL
LIN {X 0,Y 589.498,Z 481.49,A -85,B 0,C 180,E1 26593.238,E2 26593.238} C_VEL
LIN {X 0,Y 597.453,Z 495.225,A -85,B 0,C 180,E1 26592.35,E2 26592.35} C_VEL
LIN {X 0,Y 591.251,Z 743.196,A -85,B 0,C 180,E1 26588.926,E2 26588.926} C_VEL
LIN {X 0,Y 588.737,Z 843.802,A -85,B 0,C 180,E1 26587.522,E2 26587.522} C_VEL
LIN {X 0,Y 587.417,Z 869.03,A -85,B 0,C 180,E1 26587.006,E2 26587.006} C_VEL
LIN {X 0,Y 585.957,Z 890.567,A -85,B 0,C 180,E1 26586.419,E2 26586.419} C_VEL
LIN {X 0,Y 584.025,Z 914.596,A -85,B 0,C 180,E1 26585.587,E2 26585.587} C_VEL
LIN {X 0,Y 582.082,Z 935.229,A -85,B 0,C 180,E1 26584.712,E2 26584.712} C_VEL
LIN {X 0,Y 579.807,Z 957.49,A -85,B 0,C 180,E1 26583.597,E2 26583.597} C_VEL
LIN {X 0,Y 577.415,Z 978.44,A -85,B 0,C 180,E1 26582.35,E2 26582.35} C_VEL
LIN {X 0,Y 575,Z 999.285,A -85,B 0,C 180,E1 26580.921,E2 26580.921} C_VEL
LIN {X 0,Y 572.611,Z 1018.525,A -85,B 0,C 180,E1 26579.383,E2 26579.383} C_VEL
LIN {X 0,Y 570.306,Z 1037.327,A -85,B 0,C 180,E1 26577.685,E2 26577.685} C_VEL
LIN {X 0,Y 568.15,Z 1054.997,A -85,B 0,C 180,E1 26575.839,E2 26575.839} C_VEL
LIN {X 0,Y 566.195,Z 1071.782,A -85,B 0,C 180,E1 26573.854,E2 26573.854} C_VEL
LIN {X 0,Y 564.54,Z 1086.444,A -85,B 0,C 180,E1 26571.836,E2 26571.836} C_VEL
LIN {X 0,Y 563.2,Z 1099.371,A -85,B 0,C 180,E1 26569.822,E2 26569.822} C_VEL
LIN {X 0,Y 562.037,Z 1111.975,A -85,B 0,C 180,E1 26567.527,E2 26567.527} C_VEL
LIN {X 0,Y 561.309,Z 1121.114,A -85,B 0,C 180,E1 26565.604,E2 26565.604} C_VEL
LIN {X 0,Y 560.69,Z 1130.537,A -85,B 0,C 180,E1 26563.3,E2 26563.3} C_VEL
LIN {X 0,Y 560.28,Z 1138.109,A -85,B 0,C 180,E1 26561.009,E2 26561.009} C_VEL
LIN {X 0,Y 560.057,Z 1143.988,A -85,B 0,C 180,E1 26558.832,E2 26558.832} C_VEL
LIN {X 0,Y 559.954,Z 1149.188,A -85,B 0,C 180,E1 26556.253,E2 26556.253} C_VEL
LIN {X 0,Y 559.92,Z 1152.146,A -85,B 0,C 180,E1 26554.096,E2 26554.096} C_VEL
LIN {X 0,Y 559.899,Z 1154.091,A -85,B 0,C 180,E1 26551.637,E2 26551.637} C_VEL
LIN {X 0,Y 559.885,Z 1154.323,A -85,B 0,C 180,E1 26549.386,E2 26549.386} C_VEL
LIN {X 0,Y 559.89,Z 1153.429,A -85,B 0,C 180,E1 26547.339,E2 26547.339} C_VEL
LIN {X 0,Y 559.907,Z 1151.103,A -85,B 0,C 180,E1 26544.98,E2 26544.98} C_VEL
LIN {X 0,Y 559.972,Z 1147.12,A -85,B 0,C 180,E1 26542.613,E2 26542.613} C_VEL
LIN {X 0,Y 560.12,Z 1142.441,A -85,B 0,C 180,E1 26540.547,E2 26540.547} C_VEL
LIN {X 0,Y 560.403,Z 1135.598,A -85,B 0,C 180,E1 26538.159,E2 26538.159} C_VEL
LIN {X 0,Y 560.869,Z 1127.275,A -85,B 0,C 180,E1 26535.863,E2 26535.863} C_VEL
LIN {X 0,Y 561.557,Z 1117.838,A -85,B 0,C 180,E1 26533.66,E2 26533.66} C_VEL
LIN {X 0,Y 562.57,Z 1105.912,A -85,B 0,C 180,E1 26531.323,E2 26531.323} C_VEL
LIN {X 0,Y 563.74,Z 1094.151,A -85,B 0,C 180,E1 26529.331,E2 26529.331} C_VEL
LIN {X 0,Y 565.368,Z 1078.959,A -85,B 0,C 180,E1 26527.102,E2 26527.102} C_VEL
LIN {X 0,Y 567.026,Z 1064.46,A -85,B 0,C 180,E1 26525.251,E2 26525.251} C_VEL
LIN {X 0,Y 569.29,Z 1045.622,A -85,B 0,C 180,E1 26523.157,E2 26523.157} C_VEL
LIN {X 0,Y 571.349,Z 1028.765,A -85,B 0,C 180,E1 26521.517,E2 26521.517} C_VEL
LIN {X 0,Y 573.952,Z 1007.476,A -85,B 0,C 180,E1 26519.712,E2 26519.712} C_VEL
LIN {X 0,Y 576.189,Z 989.074,A -85,B 0,C 180,E1 26518.357,E2 26518.357} C_VEL
LIN {X 0,Y 578.812,Z 966.37,A -85,B 0,C 180,E1 26516.912,E2 26516.912} C_VEL
LIN {X 0,Y 580.912,Z 946.563,A -85,B 0,C 180,E1 26515.833,E2 26515.833} C_VEL
LIN {X 0,Y 583.333,Z 922.096,A -85,B 0,C 180,E1 26514.714,E2 26514.714} C_VEL
LIN {X 0,Y 585.092,Z 901.393,A -85,B 0,C 180,E1 26513.934,E2 26513.934} C_VEL
LIN {X 0,Y 586.942,Z 876.806,A -85,B 0,C 180,E1 26513.188,E2 26513.188} C_VEL
LIN {X 0,Y 588.222,Z 854.947,A -85,B 0,C 180,E1 26512.689,E2 26512.689} C_VEL
LIN {X 0,Y 589.193,Z 830.527,A -85,B 0,C 180,E1 26512.275,E2 26512.275} C_VEL
LIN {X 0,Y 594.937,Z 591.618,A -85,B 0,C 180,E1 26508.981,E2 26508.981} C_VEL
LIN {X 0,Y 597.315,Z 494.668,A -85,B 0,C 180,E1 26507.634,E2 26507.634} C_VEL
LIN {X 0,Y 581.933,Z 469.217,A -85,B 0,C 180,E1 26505.902,E2 26505.902} C_VEL
LIN {X 0,Y 575.278,Z 458.822,A -85,B 0,C 180,E1 26505.102,E2 26505.102} C_VEL
LIN {X 0,Y 567.774,Z 441.758,A -85,B 0,C 180,E1 26502.689,E2 26502.689} C_VEL
LIN {X 0,Y 562.485,Z 430.341,A -85,B 0,C 180,E1 26500.931,E2 26500.931} C_VEL
LIN {X 0,Y 561.463,Z 427.453,A -85,B 0,C 180,E1 26500.456,E2 26500.456} C_VEL
LIN {X 0,Y 561.409,Z 427.283,A -85,B 0,C 180,E1 26497.397,E2 26497.397} C_VEL
LIN {X 0,Y 561.43,Z 427.237,A -85,B 0,C 180,E1 26494.09,E2 26494.09} C_VEL
LIN {X 0,Y 561.439,Z 427.297,A -85,B 0,C 180,E1 26490.739,E2 26490.739} C_VEL
LIN {X 0,Y 561.407,Z 427.299,A -85,B 0,C 180,E1 26487.471,E2 26487.471} C_VEL
LIN {X 0,Y 561.446,Z 427.294,A -85,B 0,C 180,E1 26484.181,E2 26484.181} C_VEL
LIN {X 0,Y 561.401,Z 427.295,A -85,B 0,C 180,E1 26480.977,E2 26480.977} C_VEL
LIN {X 0,Y 561.412,Z 427.284,A -85,B 0,C 180,E1 26477.624,E2 26477.624} C_VEL
LIN {X 0,Y 561.424,Z 427.279,A -85,B 0,C 180,E1 26474.438,E2 26474.438} C_VEL
LIN {X 0,Y 561.39,Z 427.294,A -85,B 0,C 180,E1 26471.195,E2 26471.195} C_VEL
LIN {X 0,Y 561.449,Z 427.294,A -85,B 0,C 180,E1 26467.882,E2 26467.882} C_VEL
LIN {X 0,Y 561.384,Z 427.288,A -85,B 0,C 180,E1 26464.7,E2 26464.7} C_VEL
LIN {X 0,Y 561.395,Z 427.28,A -85,B 0,C 180,E1 26461.327,E2 26461.327} C_VEL
LIN {X 0,Y 561.391,Z 427.299,A -85,B 0,C 180,E1 26458.367,E2 26458.367} C_VEL
LIN {X 0,Y 561.376,Z 427.298,A -85,B 0,C 180,E1 26454.993,E2 26454.993} C_VEL
LIN {X 0,Y 561.419,Z 427.278,A -85,B 0,C 180,E1 26451.912,E2 26451.912} C_VEL
LIN {X 0,Y 561.365,Z 427.297,A -85,B 0,C 180,E1 26448.701,E2 26448.701} C_VEL
LIN {X 0,Y 561.427,Z 427.299,A -85,B 0,C 180,E1 26445.456,E2 26445.456} C_VEL
LIN {X 0,Y 561.359,Z 427.294,A -85,B 0,C 180,E1 26442.353,E2 26442.353} C_VEL
LIN {X 0,Y 561.391,Z 427.284,A -85,B 0,C 180,E1 26439.132,E2 26439.132} C_VEL
LIN {X 0,Y 561.357,Z 427.297,A -85,B 0,C 180,E1 26436.151,E2 26436.151} C_VEL
LIN {X 0,Y 561.358,Z 427.297,A -85,B 0,C 180,E1 26432.726,E2 26432.726} C_VEL
LIN {X 0,Y 561.373,Z 427.305,A -85,B 0,C 180,E1 26429.73,E2 26429.73} C_VEL
LIN {X 0,Y 561.344,Z 427.305,A -85,B 0,C 180,E1 26426.473,E2 26426.473} C_VEL
LIN {X 0,Y 561.405,Z 427.243,A -85,B 0,C 180,E1 26423.271,E2 26423.271} C_VEL
LIN {X 0,Y 561.343,Z 427.276,A -85,B 0,C 180,E1 26420.248,E2 26420.248} C_VEL
LIN {X 0,Y 561.406,Z 427.541,A -85,B 0,C 180,E1 26418.641,E2 26418.641} C_VEL
LIN {X 0,Y 562.744,Z 430.911,A -85,B 0,C 180,E1 26418.081,E2 26418.081} C_VEL
LIN {X 0,Y 568.664,Z 444.143,A -85,B 0,C 180,E1 26416.01,E2 26416.01} C_VEL
LIN {X 0,Y 575.813,Z 461.415,A -85,B 0,C 180,E1 26413.532,E2 26413.532} C_VEL
LIN {X 0,Y 582.523,Z 478.847,A -85,B 0,C 180,E1 26411.234,E2 26411.234} C_VEL
LIN {X 0,Y 585.511,Z 487.83,A -85,B 0,C 180,E1 26410.141,E2 26410.141} C_VEL
LIN {X 0,Y 585.087,Z 494.229,A -85,B 0,C 180,E1 26409.646,E2 26409.646} C_VEL
LIN {X 0,Y 594.25,Z 538.566,A -85,B 0,C 180,E1 26408.199,E2 26408.199} C_VEL
LIN {X 0,Y 591.178,Z 686.705,A -85,B 0,C 180,E1 26406.264,E2 26406.264} C_VEL
LIN {X 0,Y 590.24,Z 694.404,A -85,B 0,C 180,E1 26406.225,E2 26406.225} C_VEL
LIN {X 0,Y 584.908,Z 714.943,A -85,B 0,C 180,E1 26406.335,E2 26406.335} C_VEL
LIN {X 0,Y 584.183,Z 721.55,A -85,B 0,C 180,E1 26406.295,E2 26406.295} C_VEL
LIN {X 0,Y 581.491,Z 847.439,A -85,B 0,C 180,E1 26404.638,E2 26404.638} C_VEL
LIN {X 0,Y 580.286,Z 871.047,A -85,B 0,C 180,E1 26404.165,E2 26404.165} C_VEL
LIN {X 0,Y 578.804,Z 892.805,A -85,B 0,C 180,E1 26403.567,E2 26403.567} C_VEL
LIN {X 0,Y 576.889,Z 914.441,A -85,B 0,C 180,E1 26402.793,E2 26402.793} C_VEL
LIN {X 0,Y 574.812,Z 934.72,A -85,B 0,C 180,E1 26401.909,E2 26401.909} C_VEL
LIN {X 0,Y 572.313,Z 955.763,A -85,B 0,C 180,E1 26400.791,E2 26400.791} C_VEL
LIN {X 0,Y 569.817,Z 975.624,A -85,B 0,C 180,E1 26399.544,E2 26399.544} C_VEL
LIN {X 0,Y 567.181,Z 994.478,A -85,B 0,C 180,E1 26398.137,E2 26398.137} C_VEL
LIN {X 0,Y 564.572,Z 1012.691,A -85,B 0,C 180,E1 26396.57,E2 26396.57} C_VEL
LIN {X 0,Y 562.179,Z 1028.974,A -85,B 0,C 180,E1 26394.931,E2 26394.931} C_VEL
LIN {X 0,Y 559.78,Z 1045.418,A -85,B 0,C 180,E1 26393.028,E2 26393.028} C_VEL
LIN {X 0,Y 557.893,Z 1058.845,A -85,B 0,C 180,E1 26391.225,E2 26391.225} C_VEL
LIN {X 0,Y 556.01,Z 1073.165,A -85,B 0,C 180,E1 26388.996,E2 26388.996} C_VEL
LIN {X 0,Y 554.679,Z 1084.249,A -85,B 0,C 180,E1 26386.98,E2 26386.98} C_VEL
LIN {X 0,Y 553.554,Z 1095.066,A -85,B 0,C 180,E1 26384.648,E2 26384.648} C_VEL
LIN {X 0,Y 552.806,Z 1104.122,A -85,B 0,C 180,E1 26382.324,E2 26382.324} C_VEL
LIN {X 0,Y 552.326,Z 1111.361,A -85,B 0,C 180,E1 26379.995,E2 26379.995} C_VEL
LIN {X 0,Y 552.07,Z 1117.283,A -85,B 0,C 180,E1 26377.598,E2 26377.598} C_VEL
LIN {X 0,Y 551.956,Z 1121.319,A -85,B 0,C 180,E1 26375.301,E2 26375.301} C_VEL
LIN {X 0,Y 551.919,Z 1124.082,A -85,B 0,C 180,E1 26372.908,E2 26372.908} C_VEL
LIN {X 0,Y 551.908,Z 1125.16,A -85,B 0,C 180,E1 26370.623,E2 26370.623} C_VEL
LIN {X 0,Y 551.909,Z 1124.87,A -85,B 0,C 180,E1 26368.235,E2 26368.235} C_VEL
LIN {X 0,Y 551.93,Z 1123.032,A -85,B 0,C 180,E1 26365.948,E2 26365.948} C_VEL
LIN {X 0,Y 552.002,Z 1119.669,A -85,B 0,C 180,E1 26363.552,E2 26363.552} C_VEL
LIN {X 0,Y 552.163,Z 1114.83,A -85,B 0,C 180,E1 26361.251,E2 26361.251} C_VEL
LIN {X 0,Y 552.532,Z 1107.971,A -85,B 0,C 180,E1 26358.765,E2 26358.765} C_VEL
LIN {X 0,Y 553.106,Z 1100.278,A -85,B 0,C 180,E1 26356.553,E2 26356.553} C_VEL
LIN {X 0,Y 554.06,Z 1090.045,A -85,B 0,C 180,E1 26354.131,E2 26354.131} C_VEL
LIN {X 0,Y 555.289,Z 1079.081,A -85,B 0,C 180,E1 26351.945,E2 26351.945} C_VEL
LIN {X 0,Y 556.86,Z 1066.51,A -85,B 0,C 180,E1 26349.833,E2 26349.833} C_VEL
LIN {X 0,Y 558.775,Z 1052.682,A -85,B 0,C 180,E1 26347.817,E2 26347.817} C_VEL
LIN {X 0,Y 560.949,Z 1037.315,A -85,B 0,C 180,E1 26345.909,E2 26345.909} C_VEL
LIN {X 0,Y 563.484,Z 1020.142,A -85,B 0,C 180,E1 26344.061,E2 26344.061} C_VEL
LIN {X 0,Y 565.874,Z 1003.689,A -85,B 0,C 180,E1 26342.536,E2 26342.536} C_VEL
LIN {X 0,Y 568.642,Z 984.02,A -85,B 0,C 180,E1 26340.967,E2 26340.967} C_VEL
LIN {X 0,Y 571.103,Z 965.733,A -85,B 0,C 180,E1 26339.719,E2 26339.719} C_VEL
LIN {X 0,Y 573.613,Z 945.133,A -85,B 0,C 180,E1 26338.529,E2 26338.529} C_VEL
LIN {X 0,Y 575.738,Z 926.109,A -85,B 0,C 180,E1 26337.603,E2 26337.603} C_VEL
LIN {X 0,Y 577.905,Z 903.131,A -85,B 0,C 180,E1 26336.688,E2 26336.688} C_VEL
LIN {X 0,Y 579.647,Z 881.542,A -85,B 0,C 180,E1 26336.009,E2 26336.009} C_VEL
LIN {X 0,Y 580.989,Z 858.91,A -85,B 0,C 180,E1 26335.479,E2 26335.479} C_VEL
LIN {X 0,Y 581.895,Z 835.935,A -85,B 0,C 180,E1 26335.099,E2 26335.099} C_VEL
LIN {X 0,Y 587.031,Z 586.633,A -85,B 0,C 180,E1 26331.841,E2 26331.841} C_VEL
LIN {X 0,Y 587.988,Z 539.066,A -85,B 0,C 180,E1 26331.198,E2 26331.198} C_VEL
LIN {X 0,Y 578.541,Z 492.86,A -85,B 0,C 180,E1 26329.63,E2 26329.63} C_VEL
LIN {X 0,Y 578.585,Z 490.518,A -85,B 0,C 180,E1 26329.423,E2 26329.423} C_VEL
LIN {X 0,Y 571.363,Z 470.75,A -85,B 0,C 180,E1 26326.866,E2 26326.866} C_VEL
LIN {X 0,Y 564.384,Z 453.468,A -85,B 0,C 180,E1 26324.411,E2 26324.411} C_VEL
LIN {X 0,Y 558.147,Z 439.273,A -85,B 0,C 180,E1 26322.206,E2 26322.206} C_VEL
LIN {X 0,Y 553.467,Z 428.457,A -85,B 0,C 180,E1 26320.384,E2 26320.384} C_VEL
LIN {X 0,Y 553.415,Z 428.256,A -85,B 0,C 180,E1 26317.509,E2 26317.509} C_VEL
LIN {X 0,Y 553.418,Z 428.269,A -85,B 0,C 180,E1 26314.062,E2 26314.062} C_VEL
LIN {X 0,Y 553.444,Z 428.278,A -85,B 0,C 180,E1 26310.991,E2 26310.991} C_VEL
LIN {X 0,Y 553.403,Z 428.282,A -85,B 0,C 180,E1 26307.785,E2 26307.785} C_VEL
LIN {X 0,Y 553.473,Z 428.272,A -85,B 0,C 180,E1 26304.552,E2 26304.552} C_VEL
LIN {X 0,Y 553.408,Z 428.282,A -85,B 0,C 180,E1 26301.406,E2 26301.406} C_VEL
LIN {X 0,Y 553.449,Z 428.284,A -85,B 0,C 180,E1 26298.104,E2 26298.104} C_VEL
LIN {X 0,Y 553.43,Z 428.291,A -85,B 0,C 180,E1 26294.973,E2 26294.973} C_VEL
LIN {X 0,Y 553.424,Z 428.284,A -85,B 0,C 180,E1 26291.569,E2 26291.569} C_VEL
LIN {X 0,Y 553.484,Z 428.266,A -85,B 0,C 180,E1 26288.414,E2 26288.414} C_VEL
LIN {X 0,Y 553.427,Z 428.289,A -85,B 0,C 180,E1 26285.287,E2 26285.287} C_VEL
LIN {X 0,Y 553.493,Z 428.282,A -85,B 0,C 180,E1 26282.071,E2 26282.071} C_VEL
LIN {X 0,Y 553.435,Z 428.268,A -85,B 0,C 180,E1 26278.965,E2 26278.965} C_VEL
LIN {X 0,Y 553.464,Z 428.277,A -85,B 0,C 180,E1 26275.648,E2 26275.648} C_VEL
LIN {X 0,Y 553.463,Z 428.288,A -85,B 0,C 180,E1 26272.526,E2 26272.526} C_VEL
LIN {X 0,Y 553.448,Z 428.281,A -85,B 0,C 180,E1 26269.17,E2 26269.17} C_VEL
LIN {X 0,Y 553.509,Z 428.263,A -85,B 0,C 180,E1 26265.885,E2 26265.885} C_VEL
LIN {X 0,Y 553.455,Z 428.279,A -85,B 0,C 180,E1 26262.657,E2 26262.657} C_VEL
LIN {X 0,Y 553.473,Z 428.283,A -85,B 0,C 180,E1 26259.262,E2 26259.262} C_VEL
LIN {X 0,Y 553.5,Z 428.287,A -85,B 0,C 180,E1 26256.017,E2 26256.017} C_VEL
LIN {X 0,Y 553.463,Z 428.288,A -85,B 0,C 180,E1 26252.685,E2 26252.685} C_VEL
LIN {X 0,Y 553.506,Z 428.286,A -85,B 0,C 180,E1 26249.374,E2 26249.374} C_VEL
LIN {X 0,Y 553.487,Z 428.223,A -85,B 0,C 180,E1 26246.017,E2 26246.017} C_VEL
LIN {X 0,Y 553.47,Z 428.27,A -85,B 0,C 180,E1 26242.626,E2 26242.626} C_VEL
LIN {X 0,Y 553.501,Z 428.485,A -85,B 0,C 180,E1 26240.397,E2 26240.397} C_VEL
LIN {X 0,Y 554.865,Z 431.814,A -85,B 0,C 180,E1 26239.824,E2 26239.824} C_VEL
LIN {X 0,Y 561.191,Z 445.465,A -85,B 0,C 180,E1 26237.662,E2 26237.662} C_VEL
LIN {X 0,Y 567.456,Z 459.667,A -85,B 0,C 180,E1 26235.627,E2 26235.627} C_VEL
LIN {X 0,Y 581.464,Z 481.625,A -85,B 0,C 180,E1 26233.938,E2 26233.938} C_VEL
LIN {X 0,Y 591.293,Z 498.369,A -85,B 0,C 180,E1 26232.811,E2 26232.811} C_VEL
LIN {X 0,Y 584.811,Z 745.557,A -85,B 0,C 180,E1 26229.366,E2 26229.366} C_VEL
LIN {X 0,Y 582.237,Z 843.733,A -85,B 0,C 180,E1 26227.981,E2 26227.981} C_VEL
LIN {X 0,Y 580.853,Z 869.065,A -85,B 0,C 180,E1 26227.46,E2 26227.46} C_VEL
LIN {X 0,Y 579.314,Z 890.785,A -85,B 0,C 180,E1 26226.862,E2 26226.862} C_VEL
LIN {X 0,Y 577.267,Z 915.024,A -85,B 0,C 180,E1 26226.011,E2 26226.011} C_VEL
LIN {X 0,Y 575.232,Z 935.668,A -85,B 0,C 180,E1 26225.125,E2 26225.125} C_VEL
LIN {X 0,Y 572.764,Z 958.484,A -85,B 0,C 180,E1 26223.962,E2 26223.962} C_VEL
LIN {X 0,Y 570.344,Z 978.693,A -85,B 0,C 180,E1 26222.741,E2 26222.741} C_VEL
LIN {X 0,Y 567.801,Z 999.445,A -85,B 0,C 180,E1 26221.298,E2 26221.298} C_VEL
LIN {X 0,Y 565.38,Z 1017.981,A -85,B 0,C 180,E1 26219.799,E2 26219.799} C_VEL
LIN {X 0,Y 562.938,Z 1036.789,A -85,B 0,C 180,E1 26218.079,E2 26218.079} C_VEL
LIN {X 0,Y 560.663,Z 1054.291,A -85,B 0,C 180,E1 26216.226,E2 26216.226} C_VEL
LIN {X 0,Y 558.675,Z 1070.358,A -85,B 0,C 180,E1 26214.308,E2 26214.308} C_VEL
LIN {X 0,Y 556.901,Z 1085.243,A -85,B 0,C 180,E1 26212.262,E2 26212.262} C_VEL
LIN {X 0,Y 555.539,Z 1097.625,A -85,B 0,C 180,E1 26210.326,E2 26210.326} C_VEL
LIN {X 0,Y 554.208,Z 1111.212,A -85,B 0,C 180,E1 26207.861,E2 26207.861} C_VEL
LIN {X 0,Y 553.392,Z 1120.769,A -85,B 0,C 180,E1 26205.833,E2 26205.833} C_VEL
LIN {X 0,Y 552.732,Z 1130.233,A -85,B 0,C 180,E1 26203.495,E2 26203.495} C_VEL
LIN {X 0,Y 552.298,Z 1137.828,A -85,B 0,C 180,E1 26201.17,E2 26201.17} C_VEL
LIN {X 0,Y 552.072,Z 1143.468,A -85,B 0,C 180,E1 26199.066,E2 26199.066} C_VEL
LIN {X 0,Y 551.957,Z 1148.629,A -85,B 0,C 180,E1 26196.553,E2 26196.553} C_VEL
LIN {X 0,Y 551.925,Z 1151.808,A -85,B 0,C 180,E1 26194.26,E2 26194.26} C_VEL
LIN {X 0,Y 551.911,Z 1153.7,A -85,B 0,C 180,E1 26191.973,E2 26191.973} C_VEL
LIN {X 0,Y 551.889,Z 1154.136,A -85,B 0,C 180,E1 26189.481,E2 26189.481} C_VEL
LIN {X 0,Y 551.895,Z 1153.286,A -85,B 0,C 180,E1 26187.404,E2 26187.404} C_VEL
LIN {X 0,Y 551.914,Z 1151.161,A -85,B 0,C 180,E1 26185.156,E2 26185.156} C_VEL
LIN {X 0,Y 551.972,Z 1147.09,A -85,B 0,C 180,E1 26182.61,E2 26182.61} C_VEL
LIN {X 0,Y 552.124,Z 1142.445,A -85,B 0,C 180,E1 26180.514,E2 26180.514} C_VEL
LIN {X 0,Y 552.417,Z 1135.655,A -85,B 0,C 180,E1 26178.092,E2 26178.092} C_VEL
LIN {X 0,Y 552.933,Z 1126.957,A -85,B 0,C 180,E1 26175.656,E2 26175.656} C_VEL
LIN {X 0,Y 553.661,Z 1117.482,A -85,B 0,C 180,E1 26173.421,E2 26173.421} C_VEL
LIN {X 0,Y 554.729,Z 1105.604,A -85,B 0,C 180,E1 26171.068,E2 26171.068} C_VEL
LIN {X 0,Y 556.018,Z 1093.273,A -85,B 0,C 180,E1 26168.959,E2 26168.959} C_VEL
LIN {X 0,Y 557.703,Z 1078.433,A -85,B 0,C 180,E1 26166.769,E2 26166.769} C_VEL
LIN {X 0,Y 559.407,Z 1064.246,A -85,B 0,C 180,E1 26164.937,E2 26164.937} C_VEL
LIN {X 0,Y 561.847,Z 1045.167,A -85,B 0,C 180,E1 26162.782,E2 26162.782} C_VEL
LIN {X 0,Y 563.996,Z 1028.526,A -85,B 0,C 180,E1 26161.14,E2 26161.14} C_VEL
LIN {X 0,Y 566.71,Z 1007.616,A -85,B 0,C 180,E1 26159.342,E2 26159.342} C_VEL
LIN {X 0,Y 569.093,Z 988.999,A -85,B 0,C 180,E1 26157.953,E2 26157.953} C_VEL
LIN {X 0,Y 571.898,Z 965.785,A -85,B 0,C 180,E1 26156.462,E2 26156.462} C_VEL
LIN {X 0,Y 574.164,Z 945.446,A -85,B 0,C 180,E1 26155.348,E2 26155.348} C_VEL
LIN {X 0,Y 576.673,Z 921.199,A -85,B 0,C 180,E1 26154.24,E2 26154.24} C_VEL
LIN {X 0,Y 578.499,Z 900.639,A -85,B 0,C 180,E1 26153.462,E2 26153.462} C_VEL
LIN {X 0,Y 580.452,Z 875.359,A -85,B 0,C 180,E1 26152.7,E2 26152.7} C_VEL
LIN {X 0,Y 581.736,Z 854.181,A -85,B 0,C 180,E1 26152.217,E2 26152.217} C_VEL
LIN {X 0,Y 582.74,Z 829.057,A -85,B 0,C 180,E1 26151.794,E2 26151.794} C_VEL
LIN {X 0,Y 588.758,Z 590.903,A -85,B 0,C 180,E1 26148.479,E2 26148.479} C_VEL
LIN {X 0,Y 591.164,Z 497.871,A -85,B 0,C 180,E1 26147.175,E2 26147.175} C_VEL
LIN {X 0,Y 576.735,Z 474.046,A -85,B 0,C 180,E1 26145.514,E2 26145.514} C_VEL
LIN {X 0,Y 567.221,Z 459.237,A -85,B 0,C 180,E1 26144.343,E2 26144.343} C_VEL
LIN {X 0,Y 560.167,Z 443.35,A -85,B 0,C 180,E1 26142.019,E2 26142.019} C_VEL
LIN {X 0,Y 554.777,Z 431.677,A -85,B 0,C 180,E1 26140.165,E2 26140.165} C_VEL
LIN {X 0,Y 553.493,Z 428.419,A -85,B 0,C 180,E1 26139.587,E2 26139.587} C_VEL
LIN {X 0,Y 553.503,Z 428.285,A -85,B 0,C 180,E1 26136.465,E2 26136.465} C_VEL
LIN {X 0,Y 553.467,Z 428.231,A -85,B 0,C 180,E1 26133.189,E2 26133.189} C_VEL
LIN {X 0,Y 553.484,Z 428.273,A -85,B 0,C 180,E1 26129.789,E2 26129.789} C_VEL
LIN {X 0,Y 553.502,Z 428.273,A -85,B 0,C 180,E1 26126.5,E2 26126.5} C_VEL
LIN {X 0,Y 553.46,Z 428.281,A -85,B 0,C 180,E1 26123.194,E2 26123.194} C_VEL
LIN {X 0,Y 553.495,Z 428.282,A -85,B 0,C 180,E1 26119.854,E2 26119.854} C_VEL
LIN {X 0,Y 553.478,Z 428.283,A -85,B 0,C 180,E1 26116.585,E2 26116.585} C_VEL
LIN {X 0,Y 553.453,Z 428.279,A -85,B 0,C 180,E1 26113.264,E2 26113.264} C_VEL
LIN {X 0,Y 553.502,Z 428.265,A -85,B 0,C 180,E1 26109.987,E2 26109.987} C_VEL
LIN {X 0,Y 553.445,Z 428.286,A -85,B 0,C 180,E1 26106.848,E2 26106.848} C_VEL
LIN {X 0,Y 553.476,Z 428.288,A -85,B 0,C 180,E1 26103.522,E2 26103.522} C_VEL
LIN {X 0,Y 553.451,Z 428.268,A -85,B 0,C 180,E1 26100.414,E2 26100.414} C_VEL
LIN {X 0,Y 553.441,Z 428.274,A -85,B 0,C 180,E1 26097.1,E2 26097.1} C_VEL
LIN {X 0,Y 553.49,Z 428.286,A -85,B 0,C 180,E1 26093.881,E2 26093.881} C_VEL
LIN {X 0,Y 553.427,Z 428.287,A -85,B 0,C 180,E1 26090.642,E2 26090.642} C_VEL
LIN {X 0,Y 553.473,Z 428.268,A -85,B 0,C 180,E1 26087.373,E2 26087.373} C_VEL
LIN {X 0,Y 553.425,Z 428.289,A -85,B 0,C 180,E1 26084.364,E2 26084.364} C_VEL
LIN {X 0,Y 553.442,Z 428.291,A -85,B 0,C 180,E1 26081.022,E2 26081.022} C_VEL
LIN {X 0,Y 553.434,Z 428.285,A -85,B 0,C 180,E1 26077.948,E2 26077.948} C_VEL
LIN {X 0,Y 553.414,Z 428.284,A -85,B 0,C 180,E1 26074.607,E2 26074.607} C_VEL
LIN {X 0,Y 553.483,Z 428.272,A -85,B 0,C 180,E1 26071.397,E2 26071.397} C_VEL
LIN {X 0,Y 553.4,Z 428.281,A -85,B 0,C 180,E1 26068.279,E2 26068.279} C_VEL
LIN {X 0,Y 553.451,Z 428.24,A -85,B 0,C 180,E1 26065.061,E2 26065.061} C_VEL
LIN {X 0,Y 553.407,Z 428.273,A -85,B 0,C 180,E1 26061.967,E2 26061.967} C_VEL
LIN {X 0,Y 553.475,Z 428.507,A -85,B 0,C 180,E1 26059.495,E2 26059.495} C_VEL
LIN {X 0,Y 560.539,Z 444.508,A -85,B 0,C 180,E1 26056.851,E2 26056.851} C_VEL
LIN {X 0,Y 567.97,Z 462.092,A -85,B 0,C 180,E1 26054.233,E2 26054.233} C_VEL
LIN {X 0,Y 574.984,Z 480.459,A -85,B 0,C 180,E1 26051.752,E2 26051.752} C_VEL
LIN {X 0,Y 578.692,Z 490.884,A -85,B 0,C 180,E1 26050.437,E2 26050.437} C_VEL
LIN {X 0,Y 578.652,Z 494.169,A -85,B 0,C 180,E1 26050.213,E2 26050.213} C_VEL
LIN {X 0,Y 588.104,Z 539.999,A -85,B 0,C 180,E1 26048.683,E2 26048.683} C_VEL
LIN {X 0,Y 584.183,Z 721.55,A -85,B 0,C 180,E1 26046.295,E2 26046.295} C_VEL
LIN {X 0,Y 583.244,Z 729.247,A -85,B 0,C 180,E1 26046.255,E2 26046.255} C_VEL
LIN {X 0,Y 577.89,Z 749.78,A -85,B 0,C 180,E1 26046.369,E2 26046.369} C_VEL
LIN {X 0,Y 577.151,Z 756.387,A -85,B 0,C 180,E1 26046.329,E2 26046.329} C_VEL
LIN {X 0,Y 575.055,Z 848.031,A -85,B 0,C 180,E1 26045.105,E2 26045.105} C_VEL
LIN {X 0,Y 573.797,Z 871.326,A -85,B 0,C 180,E1 26044.631,E2 26044.631} C_VEL
LIN {X 0,Y 572.219,Z 893.558,A -85,B 0,C 180,E1 26044.013,E2 26044.013} C_VEL
LIN {X 0,Y 570.223,Z 914.978,A -85,B 0,C 180,E1 26043.235,E2 26043.235} C_VEL
LIN {X 0,Y 567.957,Z 936.192,A -85,B 0,C 180,E1 26042.298,E2 26042.298} C_VEL
LIN {X 0,Y 565.433,Z 956.315,A -85,B 0,C 180,E1 26041.207,E2 26041.207} C_VEL
LIN {X 0,Y 562.823,Z 976.117,A -85,B 0,C 180,E1 26039.948,E2 26039.948} C_VEL
LIN {X 0,Y 560.084,Z 994.868,A -85,B 0,C 180,E1 26038.532,E2 26038.532} C_VEL
LIN {X 0,Y 557.274,Z 1013.474,A -85,B 0,C 180,E1 26036.906,E2 26036.906} C_VEL
LIN {X 0,Y 554.823,Z 1029.374,A -85,B 0,C 180,E1 26035.285,E2 26035.285} C_VEL
LIN {X 0,Y 552.3,Z 1045.79,A -85,B 0,C 180,E1 26033.358,E2 26033.358} C_VEL
LIN {X 0,Y 550.293,Z 1059.328,A -85,B 0,C 180,E1 26031.516,E2 26031.516} C_VEL
LIN {X 0,Y 548.311,Z 1073.517,A -85,B 0,C 180,E1 26029.273,E2 26029.273} C_VEL
LIN {X 0,Y 546.841,Z 1085.16,A -85,B 0,C 180,E1 26027.121,E2 26027.121} C_VEL
LIN {X 0,Y 545.702,Z 1095.413,A -85,B 0,C 180,E1 26024.864,E2 26024.864} C_VEL
LIN {X 0,Y 544.893,Z 1104.448,A -85,B 0,C 180,E1 26022.506,E2 26022.506} C_VEL
LIN {X 0,Y 544.372,Z 1111.608,A -85,B 0,C 180,E1 26020.156,E2 26020.156} C_VEL
LIN {X 0,Y 544.088,Z 1117.536,A -85,B 0,C 180,E1 26017.71,E2 26017.71} C_VEL
LIN {X 0,Y 543.964,Z 1121.556,A -85,B 0,C 180,E1 26015.379,E2 26015.379} C_VEL
LIN {X 0,Y 543.924,Z 1124.298,A -85,B 0,C 180,E1 26012.95,E2 26012.95} C_VEL
LIN {X 0,Y 543.912,Z 1125.371,A -85,B 0,C 180,E1 26010.632,E2 26010.632} C_VEL
LIN {X 0,Y 543.913,Z 1125.083,A -85,B 0,C 180,E1 26008.209,E2 26008.209} C_VEL
LIN {X 0,Y 543.936,Z 1123.251,A -85,B 0,C 180,E1 26005.889,E2 26005.889} C_VEL
LIN {X 0,Y 544.014,Z 1119.911,A -85,B 0,C 180,E1 26003.457,E2 26003.457} C_VEL
LIN {X 0,Y 544.189,Z 1115.096,A -85,B 0,C 180,E1 26001.121,E2 26001.121} C_VEL
LIN {X 0,Y 544.585,Z 1108.456,A -85,B 0,C 180,E1 25998.655,E2 25998.655} C_VEL
LIN {X 0,Y 545.197,Z 1100.834,A -85,B 0,C 180,E1 25996.416,E2 25996.416} C_VEL
LIN {X 0,Y 546.215,Z 1090.652,A -85,B 0,C 180,E1 25993.953,E2 25993.953} C_VEL
LIN {X 0,Y 547.464,Z 1080.047,A -85,B 0,C 180,E1 25991.801,E2 25991.801} C_VEL
LIN {X 0,Y 549.124,Z 1067.545,A -85,B 0,C 180,E1 25989.648,E2 25989.648} C_VEL
LIN {X 0,Y 551.123,Z 1053.816,A -85,B 0,C 180,E1 25987.604,E2 25987.604} C_VEL
LIN {X 0,Y 553.394,Z 1038.598,A -85,B 0,C 180,E1 25985.672,E2 25985.672} C_VEL
LIN {X 0,Y 555.962,Z 1022.182,A -85,B 0,C 180,E1 25983.856,E2 25983.856} C_VEL
LIN {X 0,Y 558.521,Z 1005.305,A -85,B 0,C 180,E1 25982.26,E2 25982.26} C_VEL
LIN {X 0,Y 561.335,Z 986.46,A -85,B 0,C 180,E1 25980.711,E2 25980.711} C_VEL
LIN {X 0,Y 563.946,Z 967.832,A -85,B 0,C 180,E1 25979.412,E2 25979.412} C_VEL
LIN {X 0,Y 566.681,Z 946.712,A -85,B 0,C 180,E1 25978.158,E2 25978.158} C_VEL
LIN {X 0,Y 568.882,Z 927.869,A -85,B 0,C 180,E1 25977.224,E2 25977.224} C_VEL
LIN {X 0,Y 571.161,Z 905.175,A -85,B 0,C 180,E1 25976.293,E2 25976.293} C_VEL
LIN {X 0,Y 572.935,Z 884.084,A -85,B 0,C 180,E1 25975.611,E2 25975.611} C_VEL
LIN {X 0,Y 574.497,Z 859.977,A -85,B 0,C 180,E1 25975.025,E2 25975.025} C_VEL
LIN {X 0,Y 575.415,Z 838.22,A -85,B 0,C 180,E1 25974.656,E2 25974.656} C_VEL
LIN {X 0,Y 580.85,Z 589.166,A -85,B 0,C 180,E1 25971.366,E2 25971.366} C_VEL
LIN {X 0,Y 581.87,Z 540.662,A -85,B 0,C 180,E1 25970.704,E2 25970.704} C_VEL
LIN {X 0,Y 572.465,Z 494.896,A -85,B 0,C 180,E1 25969.139,E2 25969.139} C_VEL
LIN {X 0,Y 571.12,Z 492.04,A -85,B 0,C 180,E1 25968.912,E2 25968.912} C_VEL
LIN {X 0,Y 564.16,Z 473.199,A -85,B 0,C 180,E1 25966.413,E2 25966.413} C_VEL
LIN {X 0,Y 556.895,Z 455.245,A -85,B 0,C 180,E1 25963.798,E2 25963.798} C_VEL
LIN {X 0,Y 550.615,Z 440.979,A -85,B 0,C 180,E1 25961.516,E2 25961.516} C_VEL
LIN {X 0,Y 546.708,Z 432.616,A -85,B 0,C 180,E1 25960.075,E2 25960.075} C_VEL
LIN {X 0,Y 545.508,Z 429.443,A -85,B 0,C 180,E1 25959.495,E2 25959.495} C_VEL
LIN {X 0,Y 545.474,Z 429.219,A -85,B 0,C 180,E1 25956.045,E2 25956.045} C_VEL
LIN {X 0,Y 545.529,Z 429.28,A -85,B 0,C 180,E1 25952.856,E2 25952.856} C_VEL
LIN {X 0,Y 545.466,Z 429.286,A -85,B 0,C 180,E1 25949.666,E2 25949.666} C_VEL
LIN {X 0,Y 545.524,Z 429.281,A -85,B 0,C 180,E1 25946.449,E2 25946.449} C_VEL
LIN {X 0,Y 545.476,Z 429.28,A -85,B 0,C 180,E1 25943.21,E2 25943.21} C_VEL
LIN {X 0,Y 545.481,Z 429.274,A -85,B 0,C 180,E1 25939.823,E2 25939.823} C_VEL
LIN {X 0,Y 545.514,Z 429.26,A -85,B 0,C 180,E1 25936.725,E2 25936.725} C_VEL
LIN {X 0,Y 545.481,Z 429.274,A -85,B 0,C 180,E1 25933.57,E2 25933.57} C_VEL
LIN {X 0,Y 545.549,Z 429.277,A -85,B 0,C 180,E1 25930.347,E2 25930.347} C_VEL
LIN {X 0,Y 545.485,Z 429.27,A -85,B 0,C 180,E1 25927.16,E2 25927.16} C_VEL
LIN {X 0,Y 545.525,Z 429.254,A -85,B 0,C 180,E1 25923.889,E2 25923.889} C_VEL
LIN {X 0,Y 545.51,Z 429.278,A -85,B 0,C 180,E1 25920.735,E2 25920.735} C_VEL
LIN {X 0,Y 545.505,Z 429.278,A -85,B 0,C 180,E1 25917.374,E2 25917.374} C_VEL
LIN {X 0,Y 545.562,Z 429.254,A -85,B 0,C 180,E1 25914.109,E2 25914.109} C_VEL
LIN {X 0,Y 545.504,Z 429.266,A -85,B 0,C 180,E1 25910.93,E2 25910.93} C_VEL
LIN {X 0,Y 545.546,Z 429.272,A -85,B 0,C 180,E1 25907.617,E2 25907.617} C_VEL
LIN {X 0,Y 545.524,Z 429.269,A -85,B 0,C 180,E1 25904.478,E2 25904.478} C_VEL
LIN {X 0,Y 545.52,Z 429.262,A -85,B 0,C 180,E1 25901.048,E2 25901.048} C_VEL
LIN {X 0,Y 545.569,Z 429.254,A -85,B 0,C 180,E1 25897.705,E2 25897.705} C_VEL
LIN {X 0,Y 545.533,Z 429.26,A -85,B 0,C 180,E1 25894.37,E2 25894.37} C_VEL
LIN {X 0,Y 545.532,Z 429.26,A -85,B 0,C 180,E1 25890.941,E2 25890.941} C_VEL
LIN {X 0,Y 545.561,Z 429.233,A -85,B 0,C 180,E1 25887.644,E2 25887.644} C_VEL
LIN {X 0,Y 545.534,Z 429.244,A -85,B 0,C 180,E1 25884.288,E2 25884.288} C_VEL
LIN {X 0,Y 545.602,Z 429.49,A -85,B 0,C 180,E1 25881.278,E2 25881.278} C_VEL
LIN {X 0,Y 547.137,Z 433.156,A -85,B 0,C 180,E1 25880.627,E2 25880.627} C_VEL
LIN {X 0,Y 551.985,Z 443.75,A -85,B 0,C 180,E1 25878.886,E2 25878.886} C_VEL
LIN {X 0,Y 558.392,Z 457.902,A -85,B 0,C 180,E1 25876.699,E2 25876.699} C_VEL
LIN {X 0,Y 559.719,Z 460.58,A -85,B 0,C 180,E1 25876.369,E2 25876.369} C_VEL
LIN {X 0,Y 573.666,Z 482.155,A -85,B 0,C 180,E1 25874.637,E2 25874.637} C_VEL
LIN {X 0,Y 585.173,Z 501.495,A -85,B 0,C 180,E1 25873.282,E2 25873.282} C_VEL
LIN {X 0,Y 578.407,Z 748.084,A -85,B 0,C 180,E1 25869.814,E2 25869.814} C_VEL
LIN {X 0,Y 575.773,Z 843.858,A -85,B 0,C 180,E1 25868.449,E2 25868.449} C_VEL
LIN {X 0,Y 574.32,Z 869.25,A -85,B 0,C 180,E1 25867.921,E2 25867.921} C_VEL
LIN {X 0,Y 572.695,Z 891.239,A -85,B 0,C 180,E1 25867.309,E2 25867.309} C_VEL
LIN {X 0,Y 570.544,Z 915.468,A -85,B 0,C 180,E1 25866.447,E2 25866.447} C_VEL
LIN {X 0,Y 568.416,Z 936.138,A -85,B 0,C 180,E1 25865.548,E2 25865.548} C_VEL
LIN {X 0,Y 565.716,Z 959.742,A -85,B 0,C 180,E1 25864.321,E2 25864.321} C_VEL
LIN {X 0,Y 563.306,Z 978.976,A -85,B 0,C 180,E1 25863.142,E2 25863.142} C_VEL
LIN {X 0,Y 560.535,Z 1000.322,A -85,B 0,C 180,E1 25861.631,E2 25861.631} C_VEL
LIN {X 0,Y 558.011,Z 1018.749,A -85,B 0,C 180,E1 25860.115,E2 25860.115} C_VEL
LIN {X 0,Y 555.46,Z 1037.428,A -85,B 0,C 180,E1 25858.374,E2 25858.374} C_VEL
LIN {X 0,Y 553.074,Z 1054.738,A -85,B 0,C 180,E1 25856.504,E2 25856.504} C_VEL
LIN {X 0,Y 550.876,Z 1071.579,A -85,B 0,C 180,E1 25854.447,E2 25854.447} C_VEL
LIN {X 0,Y 548.947,Z 1086.932,A -85,B 0,C 180,E1 25852.264,E2 25852.264} C_VEL
LIN {X 0,Y 547.42,Z 1100.439,A -85,B 0,C 180,E1 25850.084,E2 25850.084} C_VEL
LIN {X 0,Y 546.196,Z 1112.43,A -85,B 0,C 180,E1 25847.801,E2 25847.801} C_VEL
LIN {X 0,Y 545.308,Z 1122.792,A -85,B 0,C 180,E1 25845.528,E2 25845.528} C_VEL
LIN {X 0,Y 544.667,Z 1131.735,A -85,B 0,C 180,E1 25843.158,E2 25843.158} C_VEL
LIN {X 0,Y 544.295,Z 1138.17,A -85,B 0,C 180,E1 25841.121,E2 25841.121} C_VEL
LIN {X 0,Y 544.052,Z 1144.511,A -85,B 0,C 180,E1 25838.668,E2 25838.668} C_VEL
LIN {X 0,Y 543.955,Z 1149.047,A -85,B 0,C 180,E1 25836.226,E2 25836.226} C_VEL
LIN {X 0,Y 543.922,Z 1151.935,A -85,B 0,C 180,E1 25834.006,E2 25834.006} C_VEL
LIN {X 0,Y 543.908,Z 1153.74,A -85,B 0,C 180,E1 25831.369,E2 25831.369} C_VEL
LIN {X 0,Y 543.895,Z 1153.857,A -85,B 0,C 180,E1 25829.157,E2 25829.157} C_VEL
LIN {X 0,Y 543.891,Z 1152.864,A -85,B 0,C 180,E1 25827.049,E2 25827.049} C_VEL
LIN {X 0,Y 543.915,Z 1150.197,A -85,B 0,C 180,E1 25824.515,E2 25824.515} C_VEL
LIN {X 0,Y 543.981,Z 1146.43,A -85,B 0,C 180,E1 25822.289,E2 25822.289} C_VEL
LIN {X 0,Y 544.16,Z 1141.399,A -85,B 0,C 180,E1 25820.054,E2 25820.054} C_VEL
LIN {X 0,Y 544.549,Z 1133.57,A -85,B 0,C 180,E1 25817.379,E2 25817.379} C_VEL
LIN {X 0,Y 545.1,Z 1125.375,A -85,B 0,C 180,E1 25815.119,E2 25815.119} C_VEL
LIN {X 0,Y 546.047,Z 1114.044,A -85,B 0,C 180,E1 25812.524,E2 25812.524} C_VEL
LIN {X 0,Y 547.101,Z 1103.41,A -85,B 0,C 180,E1 25810.461,E2 25810.461} C_VEL
LIN {X 0,Y 548.62,Z 1089.833,A -85,B 0,C 180,E1 25808.173,E2 25808.173} C_VEL
LIN {X 0,Y 550.345,Z 1075.548,A -85,B 0,C 180,E1 25806.099,E2 25806.099} C_VEL
LIN {X 0,Y 552.537,Z 1058.863,A -85,B 0,C 180,E1 25803.97,E2 25803.97} C_VEL
LIN {X 0,Y 554.77,Z 1042.223,A -85,B 0,C 180,E1 25802.128,E2 25802.128} C_VEL
LIN {X 0,Y 557.343,Z 1023.712,A -85,B 0,C 180,E1 25800.32,E2 25800.32} C_VEL
LIN {X 0,Y 559.872,Z 1005.071,A -85,B 0,C 180,E1 25798.747,E2 25798.747} C_VEL
LIN {X 0,Y 562.61,Z 984.721,A -85,B 0,C 180,E1 25797.237,E2 25797.237} C_VEL
LIN {X 0,Y 565.284,Z 963.084,A -85,B 0,C 180,E1 25795.875,E2 25795.875} C_VEL
LIN {X 0,Y 567.932,Z 940.672,A -85,B 0,C 180,E1 25794.665,E2 25794.665} C_VEL
LIN {X 0,Y 570.161,Z 919.25,A -85,B 0,C 180,E1 25793.71,E2 25793.71} C_VEL
LIN {X 0,Y 572.118,Z 898.152,A -85,B 0,C 180,E1 25792.918,E2 25792.918} C_VEL
LIN {X 0,Y 574.048,Z 873.313,A -85,B 0,C 180,E1 25792.184,E2 25792.184} C_VEL
LIN {X 0,Y 575.356,Z 852.186,A -85,B 0,C 180,E1 25791.709,E2 25791.709} C_VEL
LIN {X 0,Y 576.534,Z 819.58,A -85,B 0,C 180,E1 25791.19,E2 25791.19} C_VEL
LIN {X 0,Y 582.747,Z 585.819,A -85,B 0,C 180,E1 25787.904,E2 25787.904} C_VEL
LIN {X 0,Y 585.046,Z 501.163,A -85,B 0,C 180,E1 25786.707,E2 25786.707} C_VEL
LIN {X 0,Y 571.783,Z 479.181,A -85,B 0,C 180,E1 25785.145,E2 25785.145} C_VEL
LIN {X 0,Y 559.234,Z 459.81,A -85,B 0,C 180,E1 25783.572,E2 25783.572} C_VEL
LIN {X 0,Y 552.592,Z 444.98,A -85,B 0,C 180,E1 25781.329,E2 25781.329} C_VEL
LIN {X 0,Y 548.54,Z 436.334,A -85,B 0,C 180,E1 25779.914,E2 25779.914} C_VEL
LIN {X 0,Y 545.604,Z 429.504,A -85,B 0,C 180,E1 25778.745,E2 25778.745} C_VEL
LIN {X 0,Y 545.564,Z 429.272,A -85,B 0,C 180,E1 25776.428,E2 25776.428} C_VEL
LIN {X 0,Y 545.531,Z 429.218,A -85,B 0,C 180,E1 25773.107,E2 25773.107} C_VEL
LIN {X 0,Y 545.536,Z 429.261,A -85,B 0,C 180,E1 25769.661,E2 25769.661} C_VEL
LIN {X 0,Y 545.566,Z 429.259,A -85,B 0,C 180,E1 25766.329,E2 25766.329} C_VEL
LIN {X 0,Y 545.523,Z 429.268,A -85,B 0,C 180,E1 25763.056,E2 25763.056} C_VEL
LIN {X 0,Y 545.543,Z 429.27,A -85,B 0,C 180,E1 25759.709,E2 25759.709} C_VEL
LIN {X 0,Y 545.556,Z 429.271,A -85,B 0,C 180,E1 25756.395,E2 25756.395} C_VEL
LIN {X 0,Y 545.511,Z 429.269,A -85,B 0,C 180,E1 25753.137,E2 25753.137} C_VEL
LIN {X 0,Y 545.555,Z 429.253,A -85,B 0,C 180,E1 25749.814,E2 25749.814} C_VEL
LIN {X 0,Y 545.514,Z 429.274,A -85,B 0,C 180,E1 25746.631,E2 25746.631} C_VEL
LIN {X 0,Y 545.51,Z 429.279,A -85,B 0,C 180,E1 25743.152,E2 25743.152} C_VEL
LIN {X 0,Y 545.568,Z 429.255,A -85,B 0,C 180,E1 25739.895,E2 25739.895} C_VEL
LIN {X 0,Y 545.495,Z 429.258,A -85,B 0,C 180,E1 25736.637,E2 25736.637} C_VEL
LIN {X 0,Y 545.517,Z 429.27,A -85,B 0,C 180,E1 25733.263,E2 25733.263} C_VEL
LIN {X 0,Y 545.508,Z 429.274,A -85,B 0,C 180,E1 25730.185,E2 25730.185} C_VEL
LIN {X 0,Y 545.489,Z 429.265,A -85,B 0,C 180,E1 25726.862,E2 25726.862} C_VEL
LIN {X 0,Y 545.526,Z 429.262,A -85,B 0,C 180,E1 25723.823,E2 25723.823} C_VEL
LIN {X 0,Y 545.479,Z 429.279,A -85,B 0,C 180,E1 25720.512,E2 25720.512} C_VEL
LIN {X 0,Y 545.53,Z 429.28,A -85,B 0,C 180,E1 25717.248,E2 25717.248} C_VEL
LIN {X 0,Y 545.476,Z 429.279,A -85,B 0,C 180,E1 25714.134,E2 25714.134} C_VEL
LIN {X 0,Y 545.478,Z 429.279,A -85,B 0,C 180,E1 25710.697,E2 25710.697} C_VEL
LIN {X 0,Y 545.496,Z 429.272,A -85,B 0,C 180,E1 25707.64,E2 25707.64} C_VEL
LIN {X 0,Y 545.458,Z 429.222,A -85,B 0,C 180,E1 25704.343,E2 25704.343} C_VEL
LIN {X 0,Y 545.548,Z 429.276,A -85,B 0,C 180,E1 25701.165,E2 25701.165} C_VEL
LIN {X 0,Y 545.526,Z 429.648,A -85,B 0,C 180,E1 25700.338,E2 25700.338} C_VEL
LIN {X 0,Y 547.139,Z 433.252,A -85,B 0,C 180,E1 25699.689,E2 25699.689} C_VEL
LIN {X 0,Y 554.366,Z 449.342,A -85,B 0,C 180,E1 25697.016,E2 25697.016} C_VEL
LIN {X 0,Y 561.846,Z 467.249,A -85,B 0,C 180,E1 25694.322,E2 25694.322} C_VEL
LIN {X 0,Y 568.644,Z 485.239,A -85,B 0,C 180,E1 25691.869,E2 25691.869} C_VEL
LIN {X 0,Y 571.62,Z 493.347,A -85,B 0,C 180,E1 25690.869,E2 25690.869} C_VEL
LIN {X 0,Y 572.727,Z 496.15,A -85,B 0,C 180,E1 25690.719,E2 25690.719} C_VEL
LIN {X 0,Y 581.994,Z 541.68,A -85,B 0,C 180,E1 25689.174,E2 25689.174} C_VEL
LIN {X 0,Y 577.151,Z 756.387,A -85,B 0,C 180,E1 25686.329,E2 25686.329} C_VEL
LIN {X 0,Y 576.194,Z 764.085,A -85,B 0,C 180,E1 25686.29,E2 25686.29} C_VEL
LIN {X 0,Y 570.828,Z 784.612,A -85,B 0,C 180,E1 25686.406,E2 25686.406} C_VEL
LIN {X 0,Y 570.099,Z 791.217,A -85,B 0,C 180,E1 25686.365,E2 25686.365} C_VEL
LIN {X 0,Y 568.615,Z 849.793,A -85,B 0,C 180,E1 25685.564,E2 25685.564} C_VEL
LIN {X 0,Y 567.285,Z 872.542,A -85,B 0,C 180,E1 25685.084,E2 25685.084} C_VEL
LIN {X 0,Y 565.612,Z 894.852,A -85,B 0,C 180,E1 25684.451,E2 25684.451} C_VEL
LIN {X 0,Y 563.504,Z 916.315,A -85,B 0,C 180,E1 25683.654,E2 25683.654} C_VEL
LIN {X 0,Y 561.075,Z 937.795,A -85,B 0,C 180,E1 25682.682,E2 25682.682} C_VEL
LIN {X 0,Y 558.465,Z 957.737,A -85,B 0,C 180,E1 25681.581,E2 25681.581} C_VEL
LIN {X 0,Y 555.62,Z 978.081,A -85,B 0,C 180,E1 25680.253,E2 25680.253} C_VEL
LIN {X 0,Y 552.888,Z 996.027,A -85,B 0,C 180,E1 25678.873,E2 25678.873} C_VEL
LIN {X 0,Y 549.835,Z 1015.184,A -85,B 0,C 180,E1 25677.158,E2 25677.158} C_VEL
LIN {X 0,Y 547.284,Z 1031.06,A -85,B 0,C 180,E1 25675.505,E2 25675.505} C_VEL
LIN {X 0,Y 544.7,Z 1046.967,A -85,B 0,C 180,E1 25673.589,E2 25673.589} C_VEL
LIN {X 0,Y 542.52,Z 1061.056,A -85,B 0,C 180,E1 25671.63,E2 25671.63} C_VEL
LIN {X 0,Y 540.535,Z 1074.457,A -85,B 0,C 180,E1 25669.449,E2 25669.449} C_VEL
LIN {X 0,Y 539.001,Z 1086.034,A -85,B 0,C 180,E1 25667.266,E2 25667.266} C_VEL
LIN {X 0,Y 537.802,Z 1096.158,A -85,B 0,C 180,E1 25664.977,E2 25664.977} C_VEL
LIN {X 0,Y 536.949,Z 1105.085,A -85,B 0,C 180,E1 25662.584,E2 25662.584} C_VEL
LIN {X 0,Y 536.42,Z 1111.886,A -85,B 0,C 180,E1 25660.308,E2 25660.308} C_VEL
LIN {X 0,Y 536.12,Z 1117.588,A -85,B 0,C 180,E1 25657.933,E2 25657.933} C_VEL
LIN {X 0,Y 535.973,Z 1121.632,A -85,B 0,C 180,E1 25655.567,E2 25655.567} C_VEL
LIN {X 0,Y 535.93,Z 1124.448,A -85,B 0,C 180,E1 25653.102,E2 25653.102} C_VEL
LIN {X 0,Y 535.918,Z 1125.559,A -85,B 0,C 180,E1 25650.748,E2 25650.748} C_VEL
LIN {X 0,Y 535.911,Z 1125.403,A -85,B 0,C 180,E1 25648.396,E2 25648.396} C_VEL
LIN {X 0,Y 535.939,Z 1123.585,A -85,B 0,C 180,E1 25645.935,E2 25645.935} C_VEL
LIN {X 0,Y 536.024,Z 1120.354,A -85,B 0,C 180,E1 25643.466,E2 25643.466} C_VEL
LIN {X 0,Y 536.208,Z 1115.606,A -85,B 0,C 180,E1 25641.096,E2 25641.096} C_VEL
LIN {X 0,Y 536.608,Z 1109.475,A -85,B 0,C 180,E1 25638.717,E2 25638.717} C_VEL
LIN {X 0,Y 537.267,Z 1101.542,A -85,B 0,C 180,E1 25636.328,E2 25636.328} C_VEL
LIN {X 0,Y 538.288,Z 1091.955,A -85,B 0,C 180,E1 25633.932,E2 25633.932} C_VEL
LIN {X 0,Y 539.572,Z 1081.468,A -85,B 0,C 180,E1 25631.749,E2 25631.749} C_VEL
LIN {X 0,Y 541.486,Z 1067.87,A -85,B 0,C 180,E1 25629.348,E2 25629.348} C_VEL
LIN {X 0,Y 543.471,Z 1054.899,A -85,B 0,C 180,E1 25627.386,E2 25627.386} C_VEL
LIN {X 0,Y 545.844,Z 1039.859,A -85,B 0,C 180,E1 25625.429,E2 25625.429} C_VEL
LIN {X 0,Y 548.404,Z 1024.237,A -85,B 0,C 180,E1 25623.659,E2 25623.659} C_VEL
LIN {X 0,Y 551.178,Z 1006.904,A -85,B 0,C 180,E1 25621.975,E2 25621.975} C_VEL
LIN {X 0,Y 554.033,Z 988.799,A -85,B 0,C 180,E1 25620.446,E2 25620.446} C_VEL
LIN {X 0,Y 556.804,Z 969.913,A -85,B 0,C 180,E1 25619.097,E2 25619.097} C_VEL
LIN {X 0,Y 559.501,Z 950.452,A -85,B 0,C 180,E1 25617.897,E2 25617.897} C_VEL
LIN {X 0,Y 562.049,Z 929.611,A -85,B 0,C 180,E1 25616.835,E2 25616.835} C_VEL
LIN {X 0,Y 564.368,Z 908.175,A -85,B 0,C 180,E1 25615.923,E2 25615.923} C_VEL
LIN {X 0,Y 566.322,Z 885.841,A -85,B 0,C 180,E1 25615.182,E2 25615.182} C_VEL
LIN {X 0,Y 567.982,Z 862.143,A -85,B 0,C 180,E1 25614.583,E2 25614.583} C_VEL
LIN {X 0,Y 568.969,Z 840.473,A -85,B 0,C 180,E1 25614.202,E2 25614.202} C_VEL
LIN {X 0,Y 574.661,Z 593.718,A -85,B 0,C 180,E1 25610.908,E2 25610.908} C_VEL
LIN {X 0,Y 575.809,Z 542.326,A -85,B 0,C 180,E1 25610.201,E2 25610.201} C_VEL
LIN {X 0,Y 566.937,Z 498.853,A -85,B 0,C 180,E1 25608.686,E2 25608.686} C_VEL
LIN {X 0,Y 563.031,Z 491.892,A -85,B 0,C 180,E1 25608.159,E2 25608.159} C_VEL
LIN {X 0,Y 556.416,Z 474.14,A -85,B 0,C 180,E1 25605.735,E2 25605.735} C_VEL
LIN {X 0,Y 549.432,Z 457.158,A -85,B 0,C 180,E1 25603.178,E2 25603.178} C_VEL
LIN {X 0,Y 544.274,Z 445.476,A -85,B 0,C 180,E1 25601.264,E2 25601.264} C_VEL
LIN {X 0,Y 540.721,Z 437.735,A -85,B 0,C 180,E1 25599.916,E2 25599.916} C_VEL
LIN {X 0,Y 537.612,Z 430.436,A -85,B 0,C 180,E1 25598.573,E2 25598.573} C_VEL
LIN {X 0,Y 537.534,Z 430.208,A -85,B 0,C 180,E1 25595.438,E2 25595.438} C_VEL
LIN {X 0,Y 537.535,Z 430.259,A -85,B 0,C 180,E1 25591.981,E2 25591.981} C_VEL
LIN {X 0,Y 537.568,Z 430.258,A -85,B 0,C 180,E1 25588.921,E2 25588.921} C_VEL
LIN {X 0,Y 537.527,Z 430.269,A -85,B 0,C 180,E1 25585.685,E2 25585.685} C_VEL
LIN {X 0,Y 537.594,Z 430.264,A -85,B 0,C 180,E1 25582.414,E2 25582.414} C_VEL
LIN {X 0,Y 537.541,Z 430.269,A -85,B 0,C 180,E1 25579.223,E2 25579.223} C_VEL
LIN {X 0,Y 537.548,Z 430.261,A -85,B 0,C 180,E1 25575.758,E2 25575.758} C_VEL
LIN {X 0,Y 537.577,Z 430.247,A -85,B 0,C 180,E1 25572.679,E2 25572.679} C_VEL
LIN {X 0,Y 537.546,Z 430.265,A -85,B 0,C 180,E1 25569.421,E2 25569.421} C_VEL
LIN {X 0,Y 537.618,Z 430.263,A -85,B 0,C 180,E1 25566.193,E2 25566.193} C_VEL
LIN {X 0,Y 537.559,Z 430.251,A -85,B 0,C 180,E1 25562.879,E2 25562.879} C_VEL
